(* IEC 61131-3 sources: com.logicals.lc3.webinar/usRTS_RPMControl_iSOC/src_FB_LIB_SAFE/Safe/PLCOpen (part 2) *)

(* ---- SF_GuardLocking_2.iecst ---- *)
USING logicals.web.standard.safe;

NAMESPACE logicals.web.standard.safe
NAMESPACE plcopen

TYPE
	SF_GuardLocking_2_State : UINT(
		/* Static Reset detected in state 8x01. */
		Reset_Error_0 := 16#C001,
		/* S_GuardLock and S_Guard are not TRUE although the door was not re-quested to be opened. */
		Guard_Error := 16#C010,
		/* Static Reset detected in state C410. */
		Reset_Error_1 := 16#C011,
		/* S_GuardLock and S_Guard become TRUE again after being lost (C010) */
		Guard_Return := 16#C410,
		/* Lost safety acknowledge signal. S_Guard and S_GuardLock are TRUE. */
		Safety_Lost_S_Guard_And_S_GuardLock_True := 16#C450,
		/* Lost safety acknowledge signal. At least one of the variables S_Guard or S_GuardLock is FALSE. */
		Safety_Lost_S_Guard_Or_S_GuardLock_False := 16#C050,
		/* Static Reset detected in state C420. */
		Reset_Error_2 := 16#C021,
		/* Safety acknowledge signal becomes TRUE again after being lost (Cx50). */
		Safety_Return := 16#C420,
		/* Static Reset detected in state 8433. */
		Reset_Error_3 := 16#C031,
		/* Waiting time to Unlock exceeded. */
		Unlock_Request_Error := 16#C440,
		/* Static Reset detected in state C440. */
		Reset_Error_4 := 16#C041,
		/* The function block is not active (initial state). */
		Idle := 16#0000,
		/* Guard is closed and locked. */
		Guard_Closed_And_Locked:= 16#8000,
		/* Function block was activated and initiated. S_Guard and S_GuardLock are TRUE. */
		Init_S_Guard_And_S_GuardLock_True := 16#8401,
		/* Function block was activated and initiated. At least one of the variables S_Guard or S_GuardLock is FALSE. */
		Init_S_Guard_Or_S_GuardLock_False := 16#8801,
		/* Door is closed and locked, now waiting for operator reset */
		Wait_For_Reset := 16#8430,
		/* Waiting for operator to request to open the door (unlock request). */
		Wait_For_Operator := 16#8812,
		/* Lock is released and guard is open. */
		Guard_Open_And_Unlocked := 16#8822,
		/* Lock is released but guard is closed. */
		Guard_Closed_But_Unlocked := 16#8832,
		/* S_UnlockGuard is TRUE, however the acknowledge signal S_GuardLocked is still TRUE (so waiting for acknowledge <FALSE>) */
		Wait_For_Unlocked := 16#8010
	);
END_TYPE

/* This FB controls an entrance to a hazardous area via an interlocking guard with guard locking ("four state interlock-ing"). */
FUNCTION_BLOCK SF_GuardLocking_2
	{ altName:="SF_GuardLocking_2"; bgColor:="Gold"; width:=400; }
	VAR_INPUT
		/* See 5.1.1 General Input Parameters */
		Activate : BOOL := FALSE;
		/* Variable.
		 * Monitors the guard interlocking. Can be connected to the GuardOut of the SF_Guard FB.
		 * FALSE: Guard open.
		 * TRUE: Guard closed and guarded area safe. */
		S_Guard : SAFEBOOL := SAFEBOOL_Constant#SAFEFALSE;
		/* Variable.
		 * Status of the hazardous area (EDM), e.g., based on speed moni-toring or safe time off delay.
		 * FALSE: Machine in "non-safe" state.
		 * TRUE: Machine in safe state. */
		S_SafetyActive : SAFEBOOL := SAFEBOOL_Constant#SAFEFALSE;
		/* Variable.
		 * Status of the mechanical guard locking.
		 * FALSE: Guard is not locked.
		 * TRUE: Guard is locked. */
		S_GuardLock : SAFEBOOL := SAFEBOOL_Constant#SAFEFALSE;
		/* Variable.
		 * Operator intervention - request to unlock the guard.
		 * FALSE: No request.
		 * TRUE: Request made. */
		UnlockRequest : BOOL := FALSE;
		/* See 5.1.1 General Input Parameters */
		S_StartReset : SAFEBOOL := SAFEBOOL_Constant#SAFEFALSE;
		/* See 5.1.1 General Input Parameters */
		S_AutoReset : SAFEBOOL := SAFEBOOL_Constant#SAFEFALSE;
		/* See 5.1.1 General Input Parameters.
		 * Also used to request the guard to be locked again.
		 * The quality of the signal must con-form to a manual reset device. */
		Reset : BOOL := FALSE;
	END_VAR

	VAR_OUTPUT
		/* See 5.1.2 General Output Parameters */
		Ready : BOOL := FALSE;
		/* Interface to hazardous area which must be stopped.
		 * FALSE: No safe state.
		 * TRUE: Safe state. */
		S_GuardLocked : SAFEBOOL := SAFEBOOL_Constant#SAFEFALSE;
		/* Signal to unlock the guard.
		 * FALSE: Close guard.
		 * TRUE: Unlock guard. */
		S_UnlockGuard : SAFEBOOL := SAFEBOOL_Constant#SAFEFALSE;
		/* Optional. See 5.1.2 General Output Parameters */
		SafetyDemand : BOOL := FALSE;
		/* Optional. See 5.1.2 General Output Parameters */
		ResetRequest : BOOL := FALSE;
		/* See 5.1.2 General Output Parameters */
		Error : BOOL := FALSE;
		/* See 5.1.2 General Output Parameters */
		DiagCode : WORD := 16#0000;
	END_VAR

	VAR
		R_Trig_Reset : R_TRIG;
		R_Trig_UnlockRequest : R_TRIG;
		Unlock_Waiting_Timer : TON;
	END_VAR

	R_Trig_Reset(Reset);
	R_Trig_UnlockRequest(UnlockRequest);

	IF(NOT Activate) THEN
		DiagCode := TO_WORD(SF_GuardLocking_2_State#Idle);
	ELSE
		CASE TO_UINT(DiagCode) OF
			SF_GuardLocking_2_State#Idle:
				/* IF(Activate) THEN - Active is always true here */
				IF(IS(S_Guard) AND IS(S_GuardLock)) THEN
					DiagCode := TO_WORD(SF_GuardLocking_2_State#Init_S_Guard_And_S_GuardLock_True);
				ELSE
					DiagCode := TO_WORD(SF_GuardLocking_2_State#Init_S_Guard_Or_S_GuardLock_False);
				END_IF;
			SF_GuardLocking_2_State#Init_S_Guard_And_S_GuardLock_True,
			SF_GuardLocking_2_State#Init_S_Guard_Or_S_GuardLock_False:
				IF(Reset AND NOT R_Trig_Reset.Q AND IS_NOT(S_StartReset)) THEN
					DiagCode := TO_WORD(SF_GuardLocking_2_State#Reset_Error_0);
				ELSIF(IS_NOT(S_Guard) AND UnlockRequest) THEN
					DiagCode := TO_WORD(SF_GuardLocking_2_State#Guard_Open_And_Unlocked);
				ELSIF(IS_NOT(S_Guard) AND NOT UnlockRequest) THEN
					DiagCode := TO_WORD(SF_GuardLocking_2_State#Guard_Error);
				ELSIF((R_Trig_Reset.Q OR IS(S_StartReset)) AND IS(S_Guard) AND IS(S_GuardLock)) THEN
					DiagCode := TO_WORD(SF_GuardLocking_2_State#Guard_Closed_And_Locked);
				END_IF;
			SF_GuardLocking_2_State#Reset_Error_0:
				IF(NOT Reset) THEN
					IF(IS(S_Guard) AND IS(S_GuardLock)) THEN
						DiagCode := TO_WORD(SF_GuardLocking_2_State#Init_S_Guard_And_S_GuardLock_True);
					ELSE
						DiagCode := TO_WORD(SF_GuardLocking_2_State#Init_S_Guard_Or_S_GuardLock_False);
					END_IF;
				END_IF;
			SF_GuardLocking_2_State#Guard_Open_And_Unlocked:
				IF(IS_NOT(S_SafetyActive)) THEN
					DiagCode := DetermineSafetyLost_GuardLocking_2(S_Guard, S_GuardLock);
				ELSIF(IS(S_Guard)) THEN
					DiagCode := TO_WORD(SF_GuardLocking_2_State#Guard_Closed_But_Unlocked);
				END_IF;
			SF_GuardLocking_2_State#Safety_Lost_S_Guard_And_S_GuardLock_True,
			SF_GuardLocking_2_State#Safety_Lost_S_Guard_Or_S_GuardLock_False:
				IF(IS(S_SafetyActive)) THEN
					DiagCode := TO_WORD(SF_GuardLocking_2_State#Safety_Return);
				ELSIF(R_Trig_Reset.Q AND IS(S_GuardLock) AND IS(S_Guard)) THEN
					DiagCode := TO_WORD(SF_GuardLocking_2_State#Guard_Closed_And_Locked);
				END_IF;
			SF_GuardLocking_2_State#Safety_Return:
				IF(Reset AND NOT R_Trig_Reset.Q) THEN
					DiagCode := TO_WORD(SF_GuardLocking_2_State#Reset_Error_2);
				ELSIF(IS_NOT(S_SafetyActive)) THEN
					DiagCode := DetermineSafetyLost_GuardLocking_2(S_Guard, S_GuardLock);
				ELSIF(R_Trig_Reset.Q AND (IS_NOT(S_GuardLock) OR IS_NOT(S_Guard))) THEN
					DiagCode := TO_WORD(SF_GuardLocking_2_State#Wait_For_Operator);
				ELSIF(R_Trig_Reset.Q AND IS(S_GuardLock) AND IS(S_Guard)) THEN
					DiagCode := TO_WORD(SF_GuardLocking_2_State#Guard_Closed_And_Locked);
				END_IF;
			SF_GuardLocking_2_State#Reset_Error_2:
				IF(NOT Reset) THEN
					DiagCode := TO_WORD(SF_GuardLocking_2_State#Safety_Return);
				END_IF;
			SF_GuardLocking_2_State#Guard_Closed_But_Unlocked:
				IF(IS_NOT(S_SafetyActive)) THEN
					DiagCode := DetermineSafetyLost_GuardLocking_2(S_Guard, S_GuardLock);
				ELSIF(IS_NOT(S_Guard)) THEN
					DiagCode := TO_WORD(SF_GuardLocking_2_State#Guard_Open_And_Unlocked);
				ELSIF(NOT UnlockRequest) THEN
					DiagCode := TO_WORD(SF_GuardLocking_2_State#Wait_For_Operator);
				END_IF;
			SF_GuardLocking_2_State#Wait_For_Operator:
				IF(IS_NOT(S_SafetyActive)) THEN
					DiagCode := DetermineSafetyLost_GuardLocking_2(S_Guard, S_GuardLock);
				ELSIF((IS(S_SafetyActive) AND UnlockRequest) OR IS_NOT(S_Guard)) THEN
					DiagCode := TO_WORD(SF_GuardLocking_2_State#Guard_Open_And_Unlocked);
				ELSIF(IS(S_Guard) AND IS(S_GuardLock) AND IS_NOT(S_AutoReset)) THEN
					DiagCode := TO_WORD(SF_GuardLocking_2_State#Wait_For_Reset);
				ELSIF(IS(S_Guard) AND IS(S_GuardLock) AND IS(S_AutoReset)) THEN
					DiagCode := TO_WORD(SF_GuardLocking_2_State#Guard_Closed_And_Locked);
				END_IF;
			SF_GuardLocking_2_State#Wait_For_Reset:
				IF(Reset AND NOT R_Trig_Reset.Q) THEN
					DiagCode := TO_WORD(SF_GuardLocking_2_State#Reset_Error_3);
				ELSIF(IS_NOT(S_Guard) OR IS_NOT(S_GuardLock)) THEN
					DiagCode := TO_WORD(SF_GuardLocking_2_State#Guard_Error);
				ELSIF(R_Trig_Reset.Q) THEN
					DiagCode := TO_WORD(SF_GuardLocking_2_State#Guard_Closed_And_Locked);
				ELSIF(R_Trig_UnlockRequest.Q) THEN
					DiagCode := TO_WORD(SF_GuardLocking_2_State#Wait_For_Unlocked);
				END_IF;
			SF_GuardLocking_2_State#Reset_Error_3:
				IF(NOT Reset) THEN
					DiagCode := TO_WORD(SF_GuardLocking_2_State#Wait_For_Reset);
				END_IF;
			SF_GuardLocking_2_State#Guard_Error:
				IF(IS(S_GuardLock) AND IS(S_Guard)) THEN
					DiagCode := TO_WORD(SF_GuardLocking_2_State#Guard_Return);
				END_IF;
			SF_GuardLocking_2_State#Guard_Return:
				IF(IS_NOT(S_GuardLock) OR IS_NOT(S_Guard)) THEN
					DiagCode := TO_WORD(SF_GuardLocking_2_State#Guard_Error);
				ELSIF(Reset AND NOT R_Trig_Reset.Q) THEN
					DiagCode := TO_WORD(SF_GuardLocking_2_State#Reset_Error_1);
				ELSIF(R_Trig_Reset.Q) THEN
					DiagCode := TO_WORD(SF_GuardLocking_2_State#Guard_Closed_And_Locked);
				END_IF;
			SF_GuardLocking_2_State#Reset_Error_1:
				IF(NOT Reset) THEN
					DiagCode := TO_WORD(SF_GuardLocking_2_State#Guard_Return);
				END_IF;
			SF_GuardLocking_2_State#Wait_For_Unlocked:
				Unlock_Waiting_Timer();
				IF(IS_NOT(S_SafetyActive)) THEN
					DiagCode := DetermineSafetyLost_GuardLocking_2(S_Guard, S_GuardLock);
				ELSIF(IS_NOT(S_GuardLock)) THEN
					DiagCode := TO_WORD(SF_GuardLocking_2_State#Guard_Closed_But_Unlocked);
				ELSIF(Unlock_Waiting_Timer.Q) THEN
					DiagCode := TO_WORD(SF_GuardLocking_2_State#Unlock_Request_Error);
				END_IF;
			SF_GuardLocking_2_State#Unlock_Request_Error:
				IF(Reset AND NOT R_Trig_Reset.Q) THEN
					DiagCode := TO_WORD(SF_GuardLocking_2_State#Reset_Error_4);
				ELSIF(IS_NOT(S_Guard) OR IS_NOT(S_GuardLock)) THEN
					DiagCode := TO_WORD(SF_GuardLocking_2_State#Guard_Error);
				ELSIF(R_Trig_Reset.Q AND IS(S_GuardLock) AND IS(S_Guard)) THEN
					DiagCode := TO_WORD(SF_GuardLocking_2_State#Guard_Closed_And_Locked);
				END_IF;
			SF_GuardLocking_2_State#Reset_Error_4:
				IF(NOT Reset) THEN
					DiagCode := TO_WORD(SF_GuardLocking_2_State#Unlock_Request_Error);
				END_IF;
			SF_GuardLocking_2_State#Guard_Closed_And_Locked:
				IF(IS_NOT(S_GuardLock) OR IS_NOT(S_Guard)) THEN
					DiagCode := TO_WORD(SF_GuardLocking_2_State#Guard_Error);
				ELSIF(R_Trig_UnlockRequest.Q AND IS(S_SafetyActive)) THEN
					DiagCode := TO_WORD(SF_GuardLocking_2_State#Wait_For_Unlocked);
				END_IF;
		END_CASE;
	END_IF;

	CASE TO_UINT(DiagCode) OF
		SF_GuardLocking_2_State#Reset_Error_0,
		SF_GuardLocking_2_State#Guard_Error,
		SF_GuardLocking_2_State#Reset_Error_1,
		SF_GuardLocking_2_State#Reset_Error_3:
			Unlock_Waiting_Timer(IN := FALSE);
			Ready := TRUE;
			S_GuardLocked := SAFEBOOL_Constant#SAFEFALSE;
			S_UnlockGuard := SAFEBOOL_Constant#SAFEFALSE;
			SafetyDemand := FALSE;
			ResetRequest := FALSE;
			Error := TRUE;
		SF_GuardLocking_2_State#Guard_Return:
			Unlock_Waiting_Timer(IN := FALSE);
			Ready := TRUE;
			S_GuardLocked := SAFEBOOL_Constant#SAFEFALSE;
			S_UnlockGuard := SAFEBOOL_Constant#SAFEFALSE;
			SafetyDemand := FALSE;
			ResetRequest := TRUE;
			Error := TRUE;
		SF_GuardLocking_2_State#Safety_Lost_S_Guard_And_S_GuardLock_True,
		SF_GuardLocking_2_State#Safety_Return,
		SF_GuardLocking_2_State#Unlock_Request_Error:
			Unlock_Waiting_Timer(IN := FALSE);
			Ready := TRUE;
			S_GuardLocked := SAFEBOOL_Constant#SAFEFALSE;
			S_UnlockGuard := SAFEBOOL_Constant#SAFETRUE;
			SafetyDemand := FALSE;
			ResetRequest := TRUE;
			Error := TRUE;
		SF_GuardLocking_2_State#Safety_Lost_S_Guard_Or_S_GuardLock_False,
		SF_GuardLocking_2_State#Reset_Error_2,
		SF_GuardLocking_2_State#Reset_Error_4:
			Unlock_Waiting_Timer(IN := FALSE);
			Ready := TRUE;
			S_GuardLocked := SAFEBOOL_Constant#SAFEFALSE;
			S_UnlockGuard := SAFEBOOL_Constant#SAFETRUE;
			SafetyDemand := FALSE;
			ResetRequest := FALSE;
			Error := TRUE;
		SF_GuardLocking_2_State#Idle:
			Unlock_Waiting_Timer(IN := FALSE);
			Ready := FALSE;
			S_GuardLocked := SAFEBOOL_Constant#SAFEFALSE;
			S_UnlockGuard := SAFEBOOL_Constant#SAFEFALSE;
			SafetyDemand := FALSE;
			ResetRequest := FALSE;
			Error := FALSE;
		SF_GuardLocking_2_State#Guard_Closed_And_Locked:
			Unlock_Waiting_Timer(IN := FALSE);
			Ready := TRUE;
			S_GuardLocked := SAFEBOOL_Constant#SAFETRUE;
			S_UnlockGuard := SAFEBOOL_Constant#SAFEFALSE;
			SafetyDemand := FALSE;
			ResetRequest := FALSE;
			Error := FALSE;
		SF_GuardLocking_2_State#Init_S_Guard_And_S_GuardLock_True,
		SF_GuardLocking_2_State#Wait_For_Reset:
			Unlock_Waiting_Timer(IN := FALSE);
			Ready := TRUE;
			S_GuardLocked := SAFEBOOL_Constant#SAFEFALSE;
			S_UnlockGuard := SAFEBOOL_Constant#SAFEFALSE;
			SafetyDemand := FALSE;
			ResetRequest := TRUE;
			Error := FALSE;
		SF_GuardLocking_2_State#Init_S_Guard_Or_S_GuardLock_False,
		SF_GuardLocking_2_State#Wait_For_Operator:
			Unlock_Waiting_Timer(IN := FALSE);
			Ready := TRUE;
			S_GuardLocked := SAFEBOOL_Constant#SAFEFALSE;
			S_UnlockGuard := SAFEBOOL_Constant#SAFEFALSE;
			SafetyDemand := TRUE;
			ResetRequest := FALSE;
			Error := FALSE;
		SF_GuardLocking_2_State#Guard_Open_And_Unlocked,
		SF_GuardLocking_2_State#Guard_Closed_But_Unlocked:
			Unlock_Waiting_Timer(IN := FALSE);
			Ready := TRUE;
			S_GuardLocked := SAFEBOOL_Constant#SAFEFALSE;
			S_UnlockGuard := SAFEBOOL_Constant#SAFETRUE;
			SafetyDemand := TRUE;
			ResetRequest := FALSE;
			Error := FALSE;
		SF_GuardLocking_2_State#Wait_For_Unlocked:
			Unlock_Waiting_Timer(IN := TRUE, PT := T#2s);
			Ready := TRUE;
			S_GuardLocked := SAFEBOOL_Constant#SAFEFALSE;
			S_UnlockGuard := SAFEBOOL_Constant#SAFETRUE;
			SafetyDemand := FALSE;
			ResetRequest := FALSE;
			Error := FALSE;
		ELSE
			ENO := FALSE;
	END_CASE;

	ENO := ENO AND CheckSAFEBOOL(S_Guard) AND CheckSAFEBOOL(S_SafetyActive) AND CheckSAFEBOOL(S_GuardLock) AND CheckSAFEBOOL(S_StartReset) AND CheckSAFEBOOL(S_AutoReset);

END_FUNCTION_BLOCK

FUNCTION DetermineSafetyLost_GuardLocking_2 : WORD
	VAR_INPUT
		S_Guard : SAFEBOOL;
		S_GuardLock : SAFEBOOL;
	END_VAR

	IF(IS(S_Guard) AND IS(S_GuardLock)) THEN
		DetermineSafetyLost_GuardLocking_2 := TO_WORD(SF_GuardLocking_2_State#Safety_Lost_S_Guard_And_S_GuardLock_True);
	ELSE
		DetermineSafetyLost_GuardLocking_2 := TO_WORD(SF_GuardLocking_2_State#Safety_Lost_S_Guard_Or_S_GuardLock_False);
	END_IF;
END_FUNCTION

END_NAMESPACE
END_NAMESPACE

(* ---- SF_GuardLockingSerial.iecst ---- *)
USING logicals.web.standard.safe;

NAMESPACE logicals.web.standard.safe
NAMESPACE plcopen

TYPE
	SF_GuardLockingSerial_State : UINT(
	/* Static Reset detected in state 8001. */
	Reset_Error_0 := 16#C001,
	/* S_Guard is not TRUE although the door was not requested to be opened. */
	Guard_Error := 16#C010,
	/* Static Reset detected in state C410. */
	Reset_Error_1 := 16#C011,
	/* S_Guard becomes TRUE again after being lost (C010). */
	Guard_Return := 16#C410,
	/* Lost safety acknowledge signal. S_Guard is TRUE. */
	Safety_Lost_S_Guard_True := 16#C450,
	/* Lost safety acknowledge signal. S_Guard is FALSE. */
	Safety_Lost_S_Guard_False := 16#C050,
	/* Static Reset detected in state C420. */
	Reset_Error_2 := 16#C021,
	/* Safety acknowledge signal becomes TRUE again after being lost (Cx50). */
	Safety_Return := 16#C420,
	/* Static Reset detected in state 8430. */
	Reset_Error_3 := 16#C031,
	/* Waiting time to Unlock exceeded. S_Guard is TRUE. */
	Unlock_Request_Error_S_Guard_True := 16#C440,
	/* Waiting time to Unlock exceeded. S_Guard is FALSE. */
	Unlock_Request_Error_S_Guard_False := 16#C040,
	/* Static Reset detected in state Cx40. */
	Reset_Error_4 := 16#C041,
	/* The function block is not active (initial state). */
	Idle := 16#0000,
	/* Guard is closed and locked. */
	Guard_Closed_And_Locked := 16#8000,
	/* Function block was activated and initiated. S_Guard is TRUE. */
	Init_S_Guard_True := 16#8401,
	/* Function block was activated and initiated. S_Guard is FALSE. */
	Init_S_Guard_False := 16#8801,
	/* Door is closed and locked, now waiting for operator reset */
	Wait_For_Reset := 16#8430,
	/* Waiting for operator to request to open the door (unlock request). */
	Wait_For_Operator := 16#8812,
	/* Guard is unlocked. Door can be closed or open. */
	Guard_Open_And_Or_Unlocked := 16#8822,
	/* S_UnlockGuard is TRUE, however the acknowledge signal S_GuardLocked is still TRUE (so waiting for acknowledge <FALSE>) */
	Wait_For_Unlocked := 16#8410
	);
END_TYPE

/*
 * This FB controls an entrance to a hazardous area via an interlocking guard with guard locking (four state interlock-ing).
 * The used switch does not distinguish between if the safety door is unlocked but not opened or unlocked and opened.
 * Therefore we only have the S_Guard input compared to SF_GuardLocking_2.
 */
FUNCTION_BLOCK SF_GuardLockingSerial
	{ altName:="SF_GuardLockingSerial"; bgColor:="Gold"; width:=420; }
	VAR_INPUT
		/* See 5.1.1 General Input Parameters */
		Activate : BOOl := FALSE;
		/* Variable.
		 * Monitors the guard interlocking. This can be connect to S_GuardOut from the SF_Guard FB
		 * FALSE: Guard open.
		 * TRUE: Guard closed and guarded area safe. */
		S_Guard : SAFEBOOL := SAFEBOOL_Constant#SAFEFALSE;
		/* Variable.
		 * Status of the hazardous area (EDM), e.g., based on speed moni-toring or safe time off delay.
		 * FALSE: Machine in "non-safe" state.
		 * TRUE: Machine in safe state. */
		S_SafetyActive : SAFEBOOL := SAFEBOOL_Constant#SAFEFALSE;
		/* Variable.
		 * Operator intervention  request to unlock the guard.
		 * FALSE: No request.
		 * TRUE: Request made. */
		UnlockRequest : BOOL := FALSE;
		/* See 5.1.1 General Input Parameters */
		S_StartReset : SAFEBOOL := SAFEBOOL_Constant#SAFEFALSE;
		/* See 5.1.1 General Input Parameters */
		S_AutoReset : SAFEBOOL := SAFEBOOL_Constant#SAFEFALSE;
		/* See 5.1.1 General Input Parameters.
		 * Also used to request the guard to be locked again. The quality of the signal must conform to a manual reset device. */
		Reset : BOOL := FALSE;
	END_VAR

	VAR_OUTPUT
		/* See 5.1.2 General Output Parameters */
		Ready : BOOL := FALSE;
		/* Interface to hazardous area which must be stopped.
		 * FALSE: No safe state.
		 * TRUE: Safe state. */
		S_GuardLocked : SAFEBOOL := SAFEBOOL_Constant#SAFEFALSE;
		/* Signal to unlock the guard.
		 * FALSE: Close guard.
		 * TRUE: Unlock guard. */
		S_UnlockGuard : SAFEBOOL := SAFEBOOL_Constant#SAFEFALSE;
		/* See 5.1.2 General Output Parameters */
		SafetyDemand : BOOL := FALSE;
		/* See 5.1.2 General Output Parameters */
		ResetRequest : BOOL := FALSE;
		/* See 5.1.2 General Output Parameters */
		Error : BOOL := FALSE;
		/* See 5.1.2 General Output Parameters */
		DiagCode : WORD := 16#0000;
	END_VAR

	VAR
		R_Trig_Reset : R_TRIG;
		R_Trig_UnlockRequest : R_TRIG;
		Unlock_Waiting_Timer : TON;
	END_VAR

	R_Trig_Reset(Reset);
	R_Trig_UnlockRequest(UnlockRequest);

	IF(NOT Activate) THEN
		DiagCode := TO_WORD(SF_GuardLockingSerial_State#Idle);
	ELSE
		CASE TO_UINT(DiagCode) OF
			SF_GuardLockingSerial_State#Idle:
				/* IF(Activate) THEN - Active is always true here */
				IF(IS(S_Guard)) THEN
					DiagCode := TO_WORD(SF_GuardLockingSerial_State#Init_S_Guard_True);
				ELSE
					DiagCode := TO_WORD(SF_GuardLockingSerial_State#Init_S_Guard_False);
				END_IF;
			SF_GuardLockingSerial_State#Init_S_Guard_True,
			SF_GuardLockingSerial_State#Init_S_Guard_False:
				IF(Reset AND NOT R_Trig_Reset.Q AND IS_NOT(S_StartReset)) THEN
					DiagCode := TO_WORD(SF_GuardLockingSerial_State#Reset_Error_0);
				ELSIF(IS_NOT(S_Guard) AND UnlockRequest) THEN
					DiagCode := TO_WORD(SF_GuardLockingSerial_State#Guard_Open_And_Or_Unlocked);
				ELSIF(IS_NOT(S_Guard) AND NOT UnlockRequest) THEN
					DiagCode := TO_WORD(SF_GuardLockingSerial_State#Guard_Error);
				ELSIF((R_Trig_Reset.Q OR IS(S_StartReset)) AND IS(S_Guard)) THEN
					DiagCode := TO_WORD(SF_GuardLockingSerial_State#Guard_Closed_And_Locked);
				END_IF;
			SF_GuardLockingSerial_State#Guard_Open_And_Or_Unlocked:
				IF(IS_NOT(S_SafetyActive)) THEN
					DiagCode := DetermineSafetyLost_GuardLockingSerial(S_Guard);
				ELSIF(NOT UnlockRequest) THEN
					DiagCode := TO_WORD(SF_GuardLockingSerial_State#Wait_For_Operator);
				END_IF;
			SF_GuardLockingSerial_State#Safety_Lost_S_Guard_True,
			SF_GuardLockingSerial_State#Safety_Lost_S_Guard_False:
				IF(IS(S_SafetyActive)) THEN
					DiagCode := TO_WORD(SF_GuardLockingSerial_State#Safety_Return);
				ELSIF(R_Trig_Reset.Q AND IS(S_Guard)) THEN
					DiagCode := TO_WORD(SF_GuardLockingSerial_State#Guard_Closed_And_Locked);
				END_IF;
			SF_GuardLockingSerial_State#Safety_Return:
				IF(Reset AND NOT R_Trig_Reset.Q) THEN
					DiagCode := TO_WORD(SF_GuardLockingSerial_State#Reset_Error_2);
				ELSIF(IS_NOT(S_SafetyActive)) THEN
					DiagCode := DetermineSafetyLost_GuardLockingSerial(S_Guard);
				ELSIF(R_Trig_Reset.Q AND IS_NOT(S_Guard)) THEN
					DiagCode := TO_WORD(SF_GuardLockingSerial_State#Wait_For_Operator);
				ELSIF(R_Trig_Reset.Q AND IS(S_Guard)) THEN
					DiagCode := TO_WORD(SF_GuardLockingSerial_State#Guard_Closed_And_Locked);
				END_IF;
			SF_GuardLockingSerial_State#Wait_For_Operator:
				IF(IS_NOT(S_SafetyActive)) THEN
					DiagCode := DetermineSafetyLost_GuardLockingSerial(S_Guard);
				//NOTE: This transition was adapted, because when using the original transition, transition 3 would be unreachable!
				ELSIF(IS(S_Guard) AND IS_NOT(S_AutoReset)) THEN
					DiagCode := TO_WORD(SF_GuardLockingSerial_State#Wait_For_Reset);
				ELSIF(IS(S_Guard) AND IS(S_AutoReset)) THEN
					DiagCode := TO_WORD(SF_GuardLockingSerial_State#Guard_Closed_And_Locked);
				END_IF;
			SF_GuardLockingSerial_State#Wait_For_Reset:
				IF(Reset AND NOT R_Trig_Reset.Q AND IS_NOT(S_AutoReset)) THEN
					DiagCode := TO_WORD(SF_GuardLockingSerial_State#Reset_Error_3);
				ELSIF(IS_NOT(S_Guard)) THEN
					DiagCode := TO_WORD(SF_GuardLockingSerial_State#Guard_Error);
				ELSIF(R_Trig_Reset.Q) THEN
					DiagCode := TO_WORD(SF_GuardLockingSerial_State#Guard_Closed_And_Locked);
				ELSIF(R_Trig_UnlockRequest.Q) THEN
					DiagCode := TO_WORD(SF_GuardLockingSerial_State#Wait_For_Unlocked);
				END_IF;
			SF_GuardLockingSerial_State#Wait_For_Unlocked:
				Unlock_Waiting_Timer();
				IF(IS_NOT(S_Guard)) THEN
					DiagCode := TO_WORD(SF_GuardLockingSerial_State#Guard_Open_And_Or_Unlocked);
				ELSIF(R_Trig_Reset.Q AND IS(S_Guard)) THEN
					DiagCode := TO_WORD(SF_GuardLockingSerial_State#Guard_Closed_And_Locked);
				ELSIF(Unlock_Waiting_Timer.Q) THEN
					//S_Guard can only be TRUE here -> no need to check it
					DiagCode := TO_WORD(SF_GuardLockingSerial_State#Unlock_Request_Error_S_Guard_True);
				END_IF;
			SF_GuardLockingSerial_State#Unlock_Request_Error_S_Guard_True,
			SF_GuardLockingSerial_State#Unlock_Request_Error_S_Guard_False:
				IF(Reset AND NOT R_Trig_Reset.Q AND IS_NOT(S_AutoReset)) THEN
					DiagCode := TO_WORD(SF_GuardLockingSerial_State#Reset_Error_4);
				ELSIF(R_Trig_Reset.Q AND IS(S_Guard)) THEN
					DiagCode := TO_WORD(SF_GuardLockingSerial_State#Guard_Closed_And_Locked);
				END_IF;
			SF_GuardLockingSerial_State#Guard_Closed_And_Locked:
				IF(IS_NOT(S_Guard)) THEN
					DiagCode := TO_WORD(SF_GuardLockingSerial_State#Guard_Error);
				ELSIF(R_Trig_UnlockRequest.Q AND IS(S_SafetyActive)) THEN
					DiagCode := TO_WORD(SF_GuardLockingSerial_State#Wait_For_Unlocked);
				END_IF;
			SF_GuardLockingSerial_State#Guard_Error:
				IF(IS(S_Guard)) THEN
					DiagCode := TO_WORD(SF_GuardLockingSerial_State#Guard_Return);
				END_IF;
			SF_GuardLockingSerial_State#Guard_Return:
				IF(IS_NOT(S_Guard)) THEN
					DiagCode := TO_WORD(SF_GuardLockingSerial_State#Guard_Error);
				ELSIF(Reset AND NOT R_Trig_Reset.Q) THEN
					DiagCode := TO_WORD(SF_GuardLockingSerial_State#Reset_Error_1);
				ELSIF(R_Trig_Reset.Q AND IS(S_Guard)) THEN
					DiagCode := TO_WORD(SF_GuardLockingSerial_State#Guard_Closed_And_Locked);
				END_IF;
			SF_GuardLockingSerial_State#Reset_Error_0:
				IF(NOT Reset) THEN
					IF(IS(S_Guard)) THEN
						DiagCode := TO_WORD(SF_GuardLockingSerial_State#Init_S_Guard_True);
					ELSE
						DiagCode := TO_WORD(SF_GuardLockingSerial_State#Init_S_Guard_False);
					END_IF;
				END_IF;
			SF_GuardLockingSerial_State#Reset_Error_1:
				IF(NOT Reset) THEN
					DiagCode := TO_WORD(SF_GuardLockingSerial_State#Guard_Return);
				END_IF;
			SF_GuardLockingSerial_State#Reset_Error_2:
				IF(NOT Reset) THEN
					DiagCode := TO_WORD(SF_GuardLockingSerial_State#Safety_Return);
				END_IF;
			SF_GuardLockingSerial_State#Reset_Error_3:
				IF(NOT Reset) THEN
					DiagCode := TO_WORD(SF_GuardLockingSerial_State#Wait_For_Reset);
				END_IF;
			SF_GuardLockingSerial_State#Reset_Error_4:
				IF(NOT Reset) THEN
					IF(IS(S_Guard)) THEN
						DiagCode := TO_WORD(SF_GuardLockingSerial_State#Unlock_Request_Error_S_Guard_True);
					ELSE
						DiagCode := TO_WORD(SF_GuardLockingSerial_State#Unlock_Request_Error_S_Guard_False);
					END_IF;
				END_IF;
		END_CASE;
	END_IF;

	CASE TO_UINT(DiagCode) OF
		SF_GuardLockingSerial_State#Idle:
			Unlock_Waiting_Timer(IN := FALSE);
			Ready := FALSE;
			S_GuardLocked := SAFEBOOL_Constant#SAFEFALSE;
			S_UnlockGuard := SAFEBOOL_Constant#SAFEFALSE;
			SafetyDemand := FALSE;
			ResetRequest := FALSE;
			Error := FALSE;
		SF_GuardLockingSerial_State#Guard_Closed_And_Locked:
			Unlock_Waiting_Timer(IN := FALSE);
			Ready := TRUE;
			S_GuardLocked := SAFEBOOL_Constant#SAFETRUE;
			S_UnlockGuard := SAFEBOOL_Constant#SAFEFALSE;
			SafetyDemand := FALSE;
			ResetRequest := FALSE;
			Error := FALSE;
		SF_GuardLockingSerial_State#Init_S_Guard_True,
		SF_GuardLockingSerial_State#Wait_For_Reset:
			Unlock_Waiting_Timer(IN := FALSE);
			Ready := TRUE;
			S_GuardLocked := SAFEBOOL_Constant#SAFEFALSE;
			S_UnlockGuard := SAFEBOOL_Constant#SAFEFALSE;
			SafetyDemand := FALSE;
			ResetRequest := TRUE;
			Error := FALSE;
		SF_GuardLockingSerial_State#Init_S_Guard_False,
		SF_GuardLockingSerial_State#Wait_For_Operator:
			Unlock_Waiting_Timer(IN := FALSE);
			Ready := TRUE;
			S_GuardLocked := SAFEBOOL_Constant#SAFEFALSE;
			S_UnlockGuard := SAFEBOOL_Constant#SAFEFALSE;
			SafetyDemand := TRUE;
			ResetRequest := FALSE;
			Error := FALSE;
		SF_GuardLockingSerial_State#Guard_Open_And_Or_Unlocked:
			Unlock_Waiting_Timer(IN := FALSE);
			Ready := TRUE;
			S_GuardLocked := SAFEBOOL_Constant#SAFEFALSE;
			S_UnlockGuard := SAFEBOOL_Constant#SAFETRUE;
			SafetyDemand := TRUE;
			ResetRequest := FALSE;
			Error := FALSE;
		SF_GuardLockingSerial_State#Wait_For_Unlocked:
			Unlock_Waiting_Timer(IN := TRUE, PT := T#2s);
			Ready := TRUE;
			S_GuardLocked := SAFEBOOL_Constant#SAFEFALSE;
			S_UnlockGuard := SAFEBOOL_Constant#SAFETRUE;
			SafetyDemand := FALSE;
			ResetRequest := TRUE;
			Error := FALSE;
		SF_GuardLockingSerial_State#Reset_Error_0,
		SF_GuardLockingSerial_State#Guard_Error,
		SF_GuardLockingSerial_State#Reset_Error_1,
		SF_GuardLockingSerial_State#Reset_Error_3:
			Unlock_Waiting_Timer(IN := FALSE);
			Ready := TRUE;
			S_GuardLocked := SAFEBOOL_Constant#SAFEFALSE;
			S_UnlockGuard := SAFEBOOL_Constant#SAFEFALSE;
			SafetyDemand := FALSE;
			ResetRequest := FALSE;
			Error := TRUE;
		SF_GuardLockingSerial_State#Guard_Return:
			Unlock_Waiting_Timer(IN := FALSE);
			Ready := TRUE;
			S_GuardLocked := SAFEBOOL_Constant#SAFEFALSE;
			S_UnlockGuard := SAFEBOOL_Constant#SAFEFALSE;
			SafetyDemand := FALSE;
			ResetRequest := TRUE;
			Error := TRUE;
		SF_GuardLockingSerial_State#Safety_Lost_S_Guard_True,
		SF_GuardLockingSerial_State#Safety_Return,
		SF_GuardLockingSerial_State#Unlock_Request_Error_S_Guard_True:
			 Unlock_Waiting_Timer(IN := FALSE);
			Ready := TRUE;
			S_GuardLocked := SAFEBOOL_Constant#SAFEFALSE;
			S_UnlockGuard := SAFEBOOL_Constant#SAFETRUE;
			SafetyDemand := FALSE;
			ResetRequest := TRUE;
			Error := TRUE;
		SF_GuardLockingSerial_State#Safety_Lost_S_Guard_False,
		SF_GuardLockingSerial_State#Reset_Error_2,
		SF_GuardLockingSerial_State#Unlock_Request_Error_S_Guard_False,
		SF_GuardLockingSerial_State#Reset_Error_4:
			Unlock_Waiting_Timer(IN := FALSE);
			Ready := TRUE;
			S_GuardLocked := SAFEBOOL_Constant#SAFEFALSE;
			S_UnlockGuard := SAFEBOOL_Constant#SAFETRUE;
			SafetyDemand := FALSE;
			ResetRequest := FALSE;
			Error := TRUE;
		ELSE
			ENO := FALSE;
	END_CASE;

	ENO := ENO AND CheckSAFEBOOL(S_Guard) AND CheckSAFEBOOL(S_SafetyActive) AND CheckSAFEBOOL(S_StartReset) AND CheckSAFEBOOL(S_AutoReset);
END_FUNCTION_BLOCK

FUNCTION DetermineSafetyLost_GuardLockingSerial : WORD
	VAR_INPUT
		S_Guard : SAFEBOOL;
	END_VAR

	IF(IS(S_Guard)) THEN
		DetermineSafetyLost_GuardLockingSerial := TO_WORD(SF_GuardLockingSerial_State#Safety_Lost_S_Guard_True);
	ELSE
		DetermineSafetyLost_GuardLockingSerial := TO_WORD(SF_GuardLockingSerial_State#Safety_Lost_S_Guard_False);
	END_IF;
END_FUNCTION

END_NAMESPACE
END_NAMESPACE

(* ---- SF_ModeSelector.iecst ---- *)
USING logicals.web.standard.safe;

NAMESPACE logicals.web.standard.safe
NAMESPACE plcopen

TYPE
	SF_ModeSelector_State : UINT(
	/* The FB detected that two or more S_ModeX are TRUE, e.g., short-circuit of cables. Only one S_ModeX OR no S_ModeX = TRUE */
	Error_Short_Circuit := 16#C010,
	Error_Short_Circuit_Fixed := 16#C410,

	/* The FB detected that all S_ModeX are FALSE: The period following a falling S_ModeX trigger exceeds ModeMonitorTime, e.g., open-circuit of cables. Only one S_ModeX = TRUE */
	Error_Open_Circuit := 16#C020,
	Error_Open_Circuit_Fixed := 16#C420,

	/* Static Reset signal detected in state C410. */
	Reset_Error_1 := 16#C011,
	/* Static Reset signal detected in state C420. */
	Reset_Error_2 := 16#C021,
	/* The function block is not active (initial state). */
	Idle := 16#0000,
	/* State after activation or when S_ModeX has changed (unless locked) or after Reset of an error state. */
	Mode_Changed := 16#8802,
	/* Valid mode selection, but not yet locked. */
	Mode_Selected := 16#8000,
	/* Valid mode selection is locked. */
	Mode_Locked := 16#8010
	);

	ModeState : INT(Only_One_S_ModeX := 0, No_S_ModeX := 1, More_Than_One_S_ModeX := 2);

END_TYPE

/* This function block selects the system operation mode, such as manual, automatic, semi-automatic, etc. */
FUNCTION_BLOCK SF_ModeSelector
	{ altName:="SF_ModeSelector"; bgColor:="Gold"; width:=340; }
	VAR_INPUT
		/* See Table 5.1.1 General Input Parameters */
		Activate : BOOL := FALSE;
		/* Variable or constant.
		* Input 0 from mode selector switch
		* FALSE: Mode 0 is not requested by operator.
		* TRUE: Mode 0 is requested by operator. */
		S_Mode0 : SAFEBOOL := SAFEBOOL_Constant#SAFEFALSE;
		/* Variable or constant.
		 * Input 1 from mode selector switch
		 * FALSE: Mode 1 is not requested by operator.
		 * TRUE: Mode 1 is requested by operator. */
		S_Mode1 : SAFEBOOL := SAFEBOOL_Constant#SAFEFALSE;
		/* Variable or constant.
		 * Input 2 from mode selector switch
		 * FALSE: Mode 2 is not requested by operator.
		 * TRUE: Mode 2 is requested by operator. */
		S_Mode2 : SAFEBOOL := SAFEBOOL_Constant#SAFEFALSE;
		/* Variable or constant.
		 * Input 3 from mode selector switch
		 * FALSE: Mode 3 is not requested by operator.
		 * TRUE: Mode 3 is requested by operator. */
		S_Mode3 : SAFEBOOL := SAFEBOOL_Constant#SAFEFALSE;
		/* Variable or constant.
		 * Input 4 from mode selector switch
		 * FALSE: Mode 4 is not requested by operator.
		 * TRUE: Mode 4 is requested by operator. */
		S_Mode4 : SAFEBOOL := SAFEBOOL_Constant#SAFEFALSE;
		/* Variable or constant.
		 * Input 5 from mode selector switch
		 * FALSE: Mode 5 is not requested by operator.
		 * TRUE: Mode 5 is requested by operator. */
		S_Mode5 : SAFEBOOL := SAFEBOOL_Constant#SAFEFALSE;
		/* Variable or constant.
		 * Input 6 from mode selector switch
		 * FALSE: Mode 6 is not requested by operator.
		 * TRUE: Mode 6 is requested by operator. */
		S_Mode6 : SAFEBOOL := SAFEBOOL_Constant#SAFEFALSE;
		/* Variable or constant.
		 * Input 7 from mode selector switch
		 * FALSE: Mode 7 is not requested by operator.
		 * TRUE: Mode 7 is requested by operator. */
		S_Mode7 : SAFEBOOL := SAFEBOOL_Constant#SAFEFALSE;
		/* Variable or constant.
		 * Locks the selected mode
		 * FALSE: The actual S_ModeXSel output is locked therefore a change of any S_ModeX input
		 * does not lead to a change in the S_ModeXSel output even in the event of a rising edge of Set-Mode.
		 * TRUE: The selected S_ModeXSel is not locked; a mode selec-tion change is possible. */
		S_Unlock : SAFEBOOL := SAFEBOOL_Constant#SAFEFALSE;
		/* Variable (or constant FALSE, if AutoSetMode = TRUE)
		 * Sets the selected mode
		 * Operator acknowledges the setting of a mode.
		 * Any change to new S_ModeX = TRUE leads to S_AnyModeSel/S_ModeXSel = FALSE, only a rising SetMode trigger then leads to new S_ModeXSel = TRUE. */
		S_SetMode : SAFEBOOL := SAFEBOOL_Constant#SAFEFALSE;
		/* Constant.
		 * Parameterizes the acknowledgement mode
		 * FALSE: A change in mode must be acknowledged by the operator via SetMode.
		 * TRUE: A valid change of the S_ModeX input to another S_ModeX automatically leads to a change in S_ModeXSel
		 * without operator acknowledgment via SetMode (as long as this is not locked by S_Unlock). */
		AutoSetMode : BOOL := FALSE;
		/* Constant.
		 * Maximum permissible time for changing the selection input. */
		ModeMonitorTime : TIME := T#0s;
		/* See Section 5.1.1 General Input Parameters */
		Reset : BOOL := FALSE;
	END_VAR

	VAR_OUTPUT
		/* See Section 5.1.2 General Output Parameters */
		Ready : BOOL := FALSE;
		/* Indicates that mode 0 is selected and acknowledged.
		 * FALSE: Mode 0 is not selected or not active.
		 * TRUE: Mode 0 is selected and active. */
		S_Mode0Sel : SAFEBOOL := FALSE;
		/* Indicates that mode 1 is selected and acknowledged.
		 * FALSE: Mode 1 is not selected or not active.
		 * TRUE: Mode 1 is selected and active. */
		S_Mode1Sel : SAFEBOOL := FALSE;
		/* Indicates that mode 2 is selected and acknowledged.
		 * FALSE: Mode 2 is not selected or not active.
		 * TRUE: Mode 2 is selected and active. */
		S_Mode2Sel : SAFEBOOL := FALSE;
		/* Indicates that mode 3 is selected and acknowledged.
		 * FALSE: Mode 3 is not selected or not active.
		 * TRUE: Mode 3 is selected and active. */
		S_Mode3Sel : SAFEBOOL := FALSE;
		/* Indicates that mode 4 is selected and acknowledged.
		 * FALSE: Mode 4 is not selected or not active.
		 * TRUE: Mode 4 is selected and active. */
		S_Mode4Sel : SAFEBOOL := FALSE;
		/* Indicates that mode 5 is selected and acknowledged.
		 * FALSE: Mode 5 is not selected or not active.
		 * TRUE: Mode 5 is selected and active. */
		S_Mode5Sel : SAFEBOOL := FALSE;
		/* Indicates that mode 6 is selected and acknowledged.
		 * FALSE: Mode 6 is not selected or not active.
		 * TRUE: Mode 6 is selected and active. */
		S_Mode6Sel : SAFEBOOL := FALSE;
		/* Indicates that mode 7 is selected and acknowledged.
		 * FALSE: Mode 7 is not selected or not active.
		 * TRUE: Mode 7 is selected and active. */
		S_Mode7Sel : SAFEBOOL := FALSE;
		/* Indicates that any of the 8 modes is selected and acknowledged.
		 * FALSE: No S_ModeX is selected.
		 * TRUE: One of the 8 S_ModeX is selected and active. */
		S_AnyModeSel : SAFEBOOL := FALSE;
		/* Optional. See 5.1.2 General Output Parameters */
		SafetyDemand : BOOL := FALSE;
		/* Optional. See 5.1.2 General Output Parameters */
		ResetRequest : BOOL := FALSE;
		/* See Section 5.1.2 General Output Parameters */
		Error : BOOL := FALSE;
		/* See Section 5.1.2 General Output Parameters */
		DiagCode : WORD := 16#0000;
	END_VAR

	VAR
		R_Trig_Reset : R_TRIG;
		R_Trig_S_SetMode : R_TRIG;

		ModeMonitorTimer : TON;
	END_VAR

	VAR_TEMP
		OneS_ModeChanged : BOOL;

		modeState : ModeState;
	END_VAR

	IF(NOT Activate) THEN
		DiagCode := TO_WORD(SF_ModeSelector_State#Idle);
		ModeMonitorTimer(IN := FALSE);
	ELSE

		modeState := DetermineModeState(S_Mode0, S_Mode1, S_Mode2, S_Mode3, S_Mode4, S_Mode5, S_Mode6, S_Mode7);

		ModeMonitorTimer(IN := modeState = ModeState#No_S_ModeX, PT := ModeMonitorTime);

		OneS_ModeChanged := S_Mode0 <> S_Mode0Sel OR S_Mode1 <> S_Mode1Sel OR S_Mode2 <> S_Mode2Sel OR S_Mode3 <> S_Mode3Sel OR S_Mode4 <> S_Mode4Sel OR S_Mode5 <> S_Mode5Sel OR S_Mode6 <> S_Mode6Sel OR S_Mode7 <> S_Mode7Sel;

		R_Trig_Reset(Reset);
		R_Trig_S_SetMode(IS(S_SetMode));

		CASE TO_UINT(DiagCode) OF
			SF_ModeSelector_State#Idle:
				/* IF(Activate) THEN - Active is always true here */
					DiagCode := TO_WORD(SF_ModeSelector_State#Mode_Changed);
			SF_ModeSelector_State#Mode_Changed:
				IF(modeState = ModeState#More_Than_One_S_ModeX) THEN
					DiagCode := TO_WORD(SF_ModeSelector_State#Error_Short_Circuit);
				ELSIF(ModeMonitorTimer.Q) THEN
					DiagCode := TO_WORD(SF_ModeSelector_State#Error_Open_Circuit);
				ELSIF((AutoSetMode OR R_Trig_S_SetMode.Q) AND IS(S_Unlock) AND modeState = ModeState#Only_One_S_ModeX) THEN
					DiagCode := TO_WORD(SF_ModeSelector_State#Mode_Selected);
				END_IF;
			SF_ModeSelector_State#Error_Short_Circuit, SF_ModeSelector_State#Error_Short_Circuit_Fixed:
				IF(Reset AND NOT R_Trig_Reset.Q) THEN
					DiagCode := TO_WORD(SF_ModeSelector_State#Reset_Error_1);
				ELSIF((modeState = ModeState#Only_One_S_ModeX OR modeState = ModeState#No_S_ModeX) AND R_Trig_Reset.Q) THEN
					DiagCode := TO_WORD(SF_ModeSelector_State#Mode_Changed);
				ELSE
					DiagCode := TO_WORD(DetermineErrorShortCircuit(modeState));
				END_IF;
			SF_ModeSelector_State#Error_Open_Circuit, SF_ModeSelector_State#Error_Open_Circuit_Fixed:
				IF(Reset AND NOT R_Trig_Reset.Q) THEN
					DiagCode := TO_WORD(SF_ModeSelector_State#Reset_Error_2);
				ELSIF(modeState = ModeState#Only_One_S_ModeX AND R_Trig_Reset.Q) THEN
					DiagCode := TO_WORD(SF_ModeSelector_State#Mode_Changed);
				ELSE
					DiagCode := TO_WORD(DetermineErrorOpenCircuit(modeState));
				END_IF;
			 SF_ModeSelector_State#Reset_Error_1:
				IF(NOT Reset) THEN
					DiagCode := TO_WORD(DetermineErrorShortCircuit(modeState));
				END_IF;
			SF_ModeSelector_State#Reset_Error_2:
				IF(NOT Reset) THEN
					DiagCode := TO_WORD(DetermineErrorOpenCircuit(modeState));
				END_IF;
			SF_ModeSelector_State#Mode_Selected:
				IF(modeState = ModeState#More_Than_One_S_ModeX) THEN
					DiagCode := TO_WORD(DetermineErrorShortCircuit(modeState));
				ELSIF(OneS_ModeChanged) THEN
					DiagCode := TO_WORD(SF_ModeSelector_State#Mode_Changed);
				ELSIF(IS_NOT(S_Unlock)) THEN
					DiagCode := TO_WORD(SF_ModeSelector_State#Mode_Locked);
				END_IF;
			SF_ModeSelector_State#Mode_Locked:
				IF(modeState = ModeState#More_Than_One_S_ModeX AND IS(S_Unlock)) THEN
					DiagCode := TO_WORD(DetermineErrorShortCircuit(modeState));
				ELSIF(OneS_ModeChanged AND IS(S_Unlock)) THEN
					DiagCode := TO_WORD(SF_ModeSelector_State#Mode_Changed);
				ELSIF(IS(S_Unlock)) THEN
					DiagCode := TO_WORD(SF_ModeSelector_State#Mode_Selected);
				END_IF;
		END_CASE;
	END_IF;

	CASE TO_UINT(DiagCode) OF
		SF_ModeSelector_State#Error_Short_Circuit_Fixed,
		SF_ModeSelector_State#Error_Open_Circuit_Fixed:
			Ready := TRUE;
			SafetyDemand := FALSE;
			ResetRequest := TRUE;
			Error := TRUE;
			S_AnyModeSel := SAFEBOOL_Constant#SAFEFALSE;
			S_Mode0Sel := SAFEBOOL_Constant#SAFEFALSE;
			S_Mode1Sel := SAFEBOOL_Constant#SAFEFALSE;
			S_Mode2Sel := SAFEBOOL_Constant#SAFEFALSE;
			S_Mode3Sel := SAFEBOOL_Constant#SAFEFALSE;
			S_Mode4Sel := SAFEBOOL_Constant#SAFEFALSE;
			S_Mode5Sel := SAFEBOOL_Constant#SAFEFALSE;
			S_Mode6Sel := SAFEBOOL_Constant#SAFEFALSE;
			S_Mode7Sel := SAFEBOOL_Constant#SAFEFALSE;
		SF_ModeSelector_State#Error_Short_Circuit,
		SF_ModeSelector_State#Error_Open_Circuit,
		SF_ModeSelector_State#Reset_Error_1,
		SF_ModeSelector_State#Reset_Error_2:
			Ready := TRUE;
			SafetyDemand := FALSE;
			ResetRequest := FALSE;
			Error := TRUE;
			S_AnyModeSel := SAFEBOOL_Constant#SAFEFALSE;
			S_Mode0Sel := SAFEBOOL_Constant#SAFEFALSE;
			S_Mode1Sel := SAFEBOOL_Constant#SAFEFALSE;
			S_Mode2Sel := SAFEBOOL_Constant#SAFEFALSE;
			S_Mode3Sel := SAFEBOOL_Constant#SAFEFALSE;
			S_Mode4Sel := SAFEBOOL_Constant#SAFEFALSE;
			S_Mode5Sel := SAFEBOOL_Constant#SAFEFALSE;
			S_Mode6Sel := SAFEBOOL_Constant#SAFEFALSE;
			S_Mode7Sel := SAFEBOOL_Constant#SAFEFALSE;
		SF_ModeSelector_State#Idle:
			Ready := FALSE;
			SafetyDemand := FALSE;
			ResetRequest := FALSE;
			Error := FALSE;
			S_AnyModeSel := SAFEBOOL_Constant#SAFEFALSE;
			S_Mode0Sel := SAFEBOOL_Constant#SAFEFALSE;
			S_Mode1Sel := SAFEBOOL_Constant#SAFEFALSE;
			S_Mode2Sel := SAFEBOOL_Constant#SAFEFALSE;
			S_Mode3Sel := SAFEBOOL_Constant#SAFEFALSE;
			S_Mode4Sel := SAFEBOOL_Constant#SAFEFALSE;
			S_Mode5Sel := SAFEBOOL_Constant#SAFEFALSE;
			S_Mode6Sel := SAFEBOOL_Constant#SAFEFALSE;
			S_Mode7Sel := SAFEBOOL_Constant#SAFEFALSE;
		SF_ModeSelector_State#Mode_Changed:
			Ready := TRUE;
			SafetyDemand := TRUE;
			ResetRequest := FALSE;
			Error := FALSE;
			S_AnyModeSel := SAFEBOOL_Constant#SAFEFALSE;
			S_Mode0Sel := SAFEBOOL_Constant#SAFEFALSE;
			S_Mode1Sel := SAFEBOOL_Constant#SAFEFALSE;
			S_Mode2Sel := SAFEBOOL_Constant#SAFEFALSE;
			S_Mode3Sel := SAFEBOOL_Constant#SAFEFALSE;
			S_Mode4Sel := SAFEBOOL_Constant#SAFEFALSE;
			S_Mode5Sel := SAFEBOOL_Constant#SAFEFALSE;
			S_Mode6Sel := SAFEBOOL_Constant#SAFEFALSE;
			S_Mode7Sel := SAFEBOOL_Constant#SAFEFALSE;
		SF_ModeSelector_State#Mode_Selected:
			Ready := TRUE;
			SafetyDemand := FALSE;
			ResetRequest := FALSE;
			Error := FALSE;
			S_AnyModeSel := SAFEBOOL_Constant#SAFETRUE;
			S_Mode0Sel := S_Mode0;
			S_Mode1Sel := S_Mode1;
			S_Mode2Sel := S_Mode2;
			S_Mode3Sel := S_Mode3;
			S_Mode4Sel := S_Mode4;
			S_Mode5Sel := S_Mode5;
			S_Mode6Sel := S_Mode6;
			S_Mode7Sel := S_Mode7;
		SF_ModeSelector_State#Mode_Locked:
			Ready := TRUE;
			SafetyDemand := FALSE;
			ResetRequest := FALSE;
			Error := FALSE;
			S_AnyModeSel := SAFEBOOL_Constant#SAFETRUE;
	END_CASE;

	ENO := ENO AND CheckSAFEBOOL(S_Mode0) AND CheckSAFEBOOL(S_Mode1) AND CheckSAFEBOOL(S_Mode2) AND CheckSAFEBOOL(S_Mode3) AND CheckSAFEBOOL(S_Mode4) AND CheckSAFEBOOL(S_Mode5) AND CheckSAFEBOOL(S_Mode6) AND CheckSAFEBOOL(S_Mode7) AND CheckSAFEBOOL(S_Unlock) AND CheckSAFEBOOL(S_SetMode);

END_FUNCTION_BLOCK

FUNCTION DetermineModeState : INT

	VAR_INPUT
		S_Mode0 : SAFEBOOL;
		S_Mode1 : SAFEBOOL;
		S_Mode2 : SAFEBOOL;
		S_Mode3 : SAFEBOOL;
		S_Mode4 : SAFEBOOL;
		S_Mode5 : SAFEBOOL;
		S_Mode6 : SAFEBOOL;
		S_Mode7 : SAFEBOOL;
	END_VAR

	IF(XOR(IS(S_Mode0),IS(S_Mode1),IS(S_Mode2),IS(S_Mode3),IS(S_Mode4),IS(S_Mode5),IS(S_Mode6),IS(S_Mode7))) THEN
		DetermineModeState := ModeState#Only_One_S_ModeX;
	ELSIF(NOT OR(IS(S_Mode0),IS(S_Mode1),IS(S_Mode2),IS(S_Mode3),IS(S_Mode4),IS(S_Mode5),IS(S_Mode6),IS(S_Mode7))) THEN
		DetermineModeState := ModeState#No_S_ModeX;
	ELSE
		DetermineModeState := ModeState#More_Than_One_S_ModeX;
	END_IF;
END_FUNCTION

FUNCTION DetermineErrorShortCircuit : UINT
	VAR_INPUT
		modeState : ModeState;
	END_VAR

	IF(modeState = ModeState#Only_One_S_ModeX OR modeState = ModeState#No_S_ModeX) THEN
		DetermineErrorShortCircuit := SF_ModeSelector_State#Error_Short_Circuit_Fixed;
	ELSE
		DetermineErrorShortCircuit := SF_ModeSelector_State#Error_Short_Circuit;
	END_IF;
END_FUNCTION

FUNCTION DetermineErrorOpenCircuit : UINT
	VAR_INPUT
		modeState : ModeState;
	END_VAR

	IF(modeState = ModeState#Only_One_S_ModeX) THEN
		DetermineErrorOpenCircuit := SF_ModeSelector_State#Error_Open_Circuit_Fixed;
	ELSE
		DetermineErrorOpenCircuit := SF_ModeSelector_State#Error_Open_Circuit;
	END_IF;
END_FUNCTION

END_NAMESPACE
END_NAMESPACE

(* ---- SF_MutingPar_2Sensor.iecst ---- *)
USING logicals.web.standard.safe;

NAMESPACE logicals.web.standard.safe
NAMESPACE plcopen

TYPE
	SF_MutingPar_2Sensor_State : UINT(
	/* Static Reset condition detected after FB activation in state 8401. */
	Reset_Error_1 := 16#C001,
	/* Static Reset condition detected in state 8402. */
	Reset_Error_2 := 16#C011,
	/* Error detected in muting sequence state 8000, 8010, 8310. */
	Error_Muting_Sequence_Base := 16#C004,
	/* DiscTimeEntry or MaxMutingTime value out of range. */
	Parameter_Error := 16#C010,
	/* Timing error: Active muting time (when S_MutingActive = TRUE) ex-ceeds MaxMutingTime. */
	Error_Timer_MaxMuting := 16#C020,
	/* Timing error: Discrepancy time for switching MutingSwitch11 and MutingSwitch12 from FALSE to TRUE > DiscTimeEntry. */
	Error_Timer_Entry := 16#C030,
	/* The function block is not active (initial state). */
	Idle := 16#0000,
	/* Muting not active and no safety demand from AOPD. If timers from subsequent muting are still running, they are stopped. */
	AOPD_Free := 16#8000,
	/* Function block was activated. */
	Init := 16#8401,
	/* Safety demand detected by AOPD, muting not active. */
	Safety_Demand_AOPD := 16#8802,
	/* Safety demand or errors have been detected and are now cleared. Operator acknowledgment by Reset required. */
	Wait_For_Reset := 16#8402,
	/* Safety function activated. */
	Safe := 16#8804,
	/* Muting sequence is in starting phase after rising trigger of MutingSwitch11. Monitoring of DiscTimeEntry is activated. */
	Muting_Start_1 := 16#8010,
	/* Muting sequence is in starting phase after rising trigger of MutingSwitch12. Monitoring of DiscTimeEntry is activated. */
	Muting_Start_2 := 16#8310,
	/* Muting sequence is active either:
	 * - After rising trigger of the second MutingSwitch 12 or 11 has been detected.
	 * - When both MutingSwitch 11 and 12 have been actuated in the same cycle.
	 * Monitoring of DiscTimeEntry is stopped. Monitoring of MaxMutingTime is activated.
	 */
	Muting_Active := 16#8020
	);
END_TYPE

/* Muting is the intended suppression of the safety function. In this FB, parallel muting with two muting sensors is specified. */
FUNCTION_BLOCK SF_MutingPar_2Sensor
	{ altName:="SF_MutingPar_2Sensor"; bgColor:="Gold"; width:=420; }
	VAR_INPUT
		/* See Section 5.1.1 General Input Parameters */
		Activate : BOOL := FALSE;
		/* Variable.
		 * OSSD signal from AOPD.
		 * FALSE: Protection field interrupted.
		 * TRUE: Protection field not interrupted. */
		S_AOPD_In : SAFEBOOL := SAFEBOOL_Constant#SAFEFALSE;
		/* Variable.
		 * Status of Muting sensor 11.
		 * FALSE: Muting sensor 11 not actuated.
		 * TRUE: Workpiece actuates muting sensor 11.
		 * Depending on the safety requirements it can be necessary to connect a SAFEBOOL. */
		MutingSwitch11 : BOOL := FALSE;
		/* Variable.
		 * Status of Muting sensor 12.
		 * FALSE: Muting sensor 12 not actuated.
		 * TRUE: Workpiece actuates muting sensor 12.
		 * Depending on the safety requirements it can be necessary to connect a SAFEBOOL. */
		MutingSwitch12 : BOOL := FALSE;
		/* Constant 0..4 s;
		 * Max. discrepancy time for S_MutingSwitch11 and S_MutingSwitch12 entering muting gate */
		DiscTimeEntry : TIME := T#0s;
		/* Constant 0..120 min;
		 * Maximum time for complete muting sequence, timer started when both muting sensors are actuated. */
		MaxMutingTime : TIME := T#0s;
		/* Variable or constant.
		 * Command by the control system that enables the start of the muting function when needed by the machine cycle. After the start of the muting function, this signal can be switched off.
		 * FALSE: Muting not enabled
		 * TRUE: Start of Muting function enabled */
		MutingEnable : BOOL := FALSE;
		/* See Section 5.1.1 General Input Parameters */
		S_StartReset : SAFEBOOL := SAFEBOOL_Constant#SAFEFALSE;
		/* See Section 5.1.1 General Input Parameters */
		Reset : BOOL := FALSE;
	END_VAR

	VAR_OUTPUT
		/* See Section 5.1.2 General Output Parameters */
		Ready : BOOL := FALSE;
		/* Safety related output, indicates status of the muted guard.
		 * FALSE: AOPD protection field interrupted and muting not active.
		 * TRUE: AOPD protection field not interrupted or muting active. */
		S_AOPD_Out : SAFEBOOL := SAFEBOOL_Constant#SAFEFALSE;
		/* Indicates status of Muting process.
		 * FALSE: Muting not active.
		 * TRUE: Muting active. */
		S_MutingActive : SAFEBOOL := SAFEBOOL_Constant#SAFEFALSE;
		/* Optional. See 5.1.2 General Output Parameters */
		SafetyDemand : BOOL := FALSE;
		/* Optional. See 5.1.2 General Output Parameters */
		ResetRequest : BOOL := FALSE;
		/* See Section 5.1.2 General Output Parameters */
		Error : BOOL := FALSE;
		/* See Section 5.1.2 General Output Parameters */
		DiagCode : WORD := 16#0000;
	END_VAR

	VAR
		/* ControlCode is used for state tracking */
		ControlCode : UINT := 16#0000;
		MutingTimer : TON;
		DiscTimeEntryTimer : TON;
		R_Trig_Reset : R_TRIG;
		R_Trig_S11 : R_TRIG;
		R_Trig_S12 : R_TRIG;
	END_VAR

	R_Trig_Reset(Reset);
	R_Trig_S11(MutingSwitch11);
	R_Trig_S12(MutingSwitch12);

	IF(NOT Activate) THEN
		ControlCode := SF_MutingPar_2Sensor_State#Idle;
		DiagCode := TO_WORD(ControlCode);
	ELSE
		CASE TO_UINT(ControlCode) OF
			SF_MutingPar_2Sensor_State#Idle:
				/* IF(Activate) THEN - Active is always true here */
					ControlCode := SF_MutingPar_2Sensor_State#Init;
					DiagCode := TO_WORD(ControlCode);
			SF_MutingPar_2Sensor_State#Init:
				IF(Reset AND NOT R_Trig_Reset.Q) THEN
					ControlCode := SF_MutingPar_2Sensor_State#Reset_Error_1;
					DiagCode := TO_WORD(ControlCode);
				ELSIF(DiscTimeEntry < T#0s OR DiscTimeEntry > T#4s OR MaxMutingTime < T#0s OR MaxMutingTime > T#120m) THEN
					ControlCode := SF_MutingPar_2Sensor_State#Parameter_Error;
					DiagCode := TO_WORD(ControlCode);
				ELSIF(R_Trig_Reset.Q OR IS(S_StartReset)) THEN
					ControlCode := SF_MutingPar_2Sensor_State#Safe;
					DiagCode := TO_WORD(ControlCode);
				END_IF;
			SF_MutingPar_2Sensor_State#Safe:
				IF(IS_NOT(S_AOPD_In)) THEN
					ControlCode := SF_MutingPar_2Sensor_State#Safety_Demand_AOPD;
					DiagCode := TO_WORD(ControlCode);
				ELSE
					ControlCode := SF_MutingPar_2Sensor_State#AOPD_Free;
					DiagCode := TO_WORD(ControlCode);
				END_IF;
			SF_MutingPar_2Sensor_State#Safety_Demand_AOPD:
				IF(IS(S_AOPD_In)) THEN
					ControlCode := SF_MutingPar_2Sensor_State#Wait_For_Reset;
					DiagCode := TO_WORD(ControlCode);
				END_IF;
			SF_MutingPar_2Sensor_State#Wait_For_Reset:
				IF(Reset AND NOT R_Trig_Reset.Q) THEN
					ControlCode := SF_MutingPar_2Sensor_State#Reset_Error_2;
					DiagCode := TO_WORD(ControlCode);
				ELSIF(R_Trig_Reset.Q) THEN
					ControlCode := SF_MutingPar_2Sensor_State#Safe;
					DiagCode := TO_WORD(ControlCode);
				END_IF;
			SF_MutingPar_2Sensor_State#AOPD_Free:
				IF((R_Trig_S11.Q AND MutingSwitch12 AND NOT R_Trig_S12.Q) OR
				   (R_Trig_S12.Q AND MutingSwitch11 AND NOT R_Trig_S11.Q) OR
				   ((MutingSwitch11 AND NOT R_Trig_S11.Q) AND (MutingSwitch12 AND NOT R_Trig_S12.Q)) OR
				   (NOT MutingEnable AND R_Trig_S11.Q) OR
				   (NOT MutingEnable AND R_Trig_S12.Q )) THEN
					ControlCode := SF_MutingPar_2Sensor_State#Error_Muting_Sequence_Base;
					IF(MutingEnable) THEN
						DiagCode := TO_WORD(SF_MutingPar_2Sensor_State#Error_Muting_Sequence_Base + GetErrorStateOfMutingSensors(MutingSwitch11, MutingSwitch12));
					ELSE
						DiagCode := TO_WORD(SF_MutingPar_2Sensor_State#Error_Muting_Sequence_Base + 16#0F00 + GetErrorStateOfMutingSensors(MutingSwitch11, MutingSwitch12));
					END_IF;
				ELSIF(IS_NOT(S_AOPD_In)) THEN
					ControlCode := SF_MutingPar_2Sensor_State#Safety_Demand_AOPD;
					DiagCode := TO_WORD(ControlCode);
				ELSIF(MutingEnable AND R_Trig_S11.Q AND NOT MutingSwitch12) THEN
					ControlCode := SF_MutingPar_2Sensor_State#Muting_Start_1;
					DiagCode := TO_WORD(ControlCode);
				ELSIF(MutingEnable AND NOT MutingSwitch11 AND R_Trig_S12.Q) THEN
					ControlCode := SF_MutingPar_2Sensor_State#Muting_Start_2;
					DiagCode := TO_WORD(ControlCode);
				ELSIF(MutingEnable AND R_Trig_S11.Q AND R_Trig_S12.Q) THEN
					ControlCode := SF_MutingPar_2Sensor_State#Muting_Active;
					DiagCode := TO_WORD(ControlCode);
				END_IF;
			SF_MutingPar_2Sensor_State#Muting_Start_1:
				MutingTimer();
				DiscTimeEntryTimer();

				IF(NOT MutingEnable OR NOT MutingSwitch11) THEN
					ControlCode := SF_MutingPar_2Sensor_State#Error_Muting_Sequence_Base;
					IF(MutingEnable) THEN
						DiagCode := TO_WORD(SF_MutingPar_2Sensor_State#Error_Muting_Sequence_Base + 16#0100 + GetErrorStateOfMutingSensors(MutingSwitch11, MutingSwitch12));
					ELSE
						DiagCode := TO_WORD(SF_MutingPar_2Sensor_State#Error_Muting_Sequence_Base + 16#0F00 + GetErrorStateOfMutingSensors(MutingSwitch11, MutingSwitch12));
					END_IF;
				ELSIF(MutingTimer.Q) THEN
					ControlCode := SF_MutingPar_2Sensor_State#Error_Timer_MaxMuting;
					DiagCode := TO_WORD(ControlCode);
				ELSIF(DiscTimeEntryTimer.Q) THEN
					ControlCode := SF_MutingPar_2Sensor_State#Error_Timer_Entry;
					DiagCode := TO_WORD(ControlCode);
				ELSIF(IS_NOT(S_AOPD_In)) THEN
					ControlCode := SF_MutingPar_2Sensor_State#Safety_Demand_AOPD;
					DiagCode := TO_WORD(ControlCode);
				ELSIF(MutingEnable AND MutingSwitch11 AND R_Trig_S12.Q) THEN
					ControlCode := SF_MutingPar_2Sensor_State#Muting_Active;
					DiagCode := TO_WORD(ControlCode);
				END_IF;
			SF_MutingPar_2Sensor_State#Muting_Start_2:
				MutingTimer();
				DiscTimeEntryTimer();

				IF(NOT MutingEnable OR NOT MutingSwitch12) THEN
					ControlCode := SF_MutingPar_2Sensor_State#Error_Muting_Sequence_Base;
					IF(MutingEnable) THEN
						DiagCode := TO_WORD(SF_MutingPar_2Sensor_State#Error_Muting_Sequence_Base + 16#0200 + GetErrorStateOfMutingSensors(MutingSwitch11, MutingSwitch12));
					ELSE
						DiagCode := TO_WORD(SF_MutingPar_2Sensor_State#Error_Muting_Sequence_Base + 16#0F00 + GetErrorStateOfMutingSensors(MutingSwitch11, MutingSwitch12));
					END_IF;
				ELSIF(MutingTimer.Q) THEN
					ControlCode := SF_MutingPar_2Sensor_State#Error_Timer_MaxMuting;
					DiagCode := TO_WORD(ControlCode);
				ELSIF(DiscTimeEntryTimer.Q) THEN
					ControlCode := SF_MutingPar_2Sensor_State#Error_Timer_Entry;
					DiagCode := TO_WORD(ControlCode);
				ELSIF(IS_NOT(S_AOPD_In)) THEN
					ControlCode := SF_MutingPar_2Sensor_State#Safety_Demand_AOPD;
					DiagCode := TO_WORD(ControlCode);
				ELSIF(MutingEnable AND R_Trig_S11.Q AND MutingSwitch12) THEN
					ControlCode := SF_MutingPar_2Sensor_State#Muting_Active;
					DiagCode := TO_WORD(ControlCode);
				END_IF;
			SF_MutingPar_2Sensor_State#Muting_Active:
				MutingTimer();
				DiscTimeEntryTimer();

				IF(MutingTimer.Q) THEN
					ControlCode := SF_MutingPar_2Sensor_State#Error_Timer_MaxMuting;
					DiagCode := TO_WORD(ControlCode);
				ELSIF(NOT MutingSwitch11 OR NOT MutingSwitch12) THEN
					ControlCode := SF_MutingPar_2Sensor_State#AOPD_Free;
					DiagCode := TO_WORD(ControlCode);
				END_IF;
			SF_MutingPar_2Sensor_State#Error_Muting_Sequence_Base:
				IF(NOT (MutingSwitch11 OR MutingSwitch12)) THEN
					ControlCode := SF_MutingPar_2Sensor_State#Wait_For_Reset;
					DiagCode := TO_WORD(ControlCode);
				END_IF;
			SF_MutingPar_2Sensor_State#Error_Timer_MaxMuting,
			SF_MutingPar_2Sensor_State#Error_Timer_Entry:
				IF(NOT (MutingSwitch11 OR MutingSwitch12)) THEN
					ControlCode := SF_MutingPar_2Sensor_State#Wait_For_Reset;
					DiagCode := TO_WORD(ControlCode);
				END_IF;
			SF_MutingPar_2Sensor_State#Reset_Error_1:
				IF(NOT Reset) THEN
					ControlCode := SF_MutingPar_2Sensor_State#Init;
					DiagCode := TO_WORD(ControlCode);
				END_IF;
			SF_MutingPar_2Sensor_State#Reset_Error_2:
				IF(NOT Reset) THEN
					ControlCode := SF_MutingPar_2Sensor_State#Wait_For_Reset;
					DiagCode := TO_WORD(ControlCode);
				END_IF;
		END_CASE;
	END_IF;

	CASE TO_UINT(ControlCode) OF
		SF_MutingPar_2Sensor_State#Idle:
			DiscTimeEntryTimer(IN := FALSE);
			MutingTimer(IN := FALSE);
			Ready := FALSE;
			S_AOPD_Out := SAFEBOOL_Constant#SAFEFALSE;
			S_MutingActive := SAFEBOOL_Constant#SAFEFALSE;
			SafetyDemand := FALSE;
			ResetRequest := FALSE;
			Error := FALSE;
		SF_MutingPar_2Sensor_State#AOPD_Free:
			DiscTimeEntryTimer(IN := FALSE);
			MutingTimer(IN := FALSE);
			Ready := TRUE;
			S_AOPD_Out := SAFEBOOL_Constant#SAFETRUE;
			S_MutingActive := SAFEBOOL_Constant#SAFEFALSE;
			SafetyDemand := FALSE;
			ResetRequest := FALSE;
			Error := FALSE;
		SF_MutingPar_2Sensor_State#Init,
		SF_MutingPar_2Sensor_State#Wait_For_Reset:
			DiscTimeEntryTimer(IN := FALSE);
			MutingTimer(IN := FALSE);
			Ready := TRUE;
			S_AOPD_Out := SAFEBOOL_Constant#SAFEFALSE;
			S_MutingActive := SAFEBOOL_Constant#SAFEFALSE;
			SafetyDemand := FALSE;
			ResetRequest := TRUE;
			Error := FALSE;
		SF_MutingPar_2Sensor_State#Safety_Demand_AOPD:
			DiscTimeEntryTimer(IN := FALSE);
			MutingTimer(IN := FALSE);
			Ready := TRUE;
			S_AOPD_Out := SAFEBOOL_Constant#SAFEFALSE;
			S_MutingActive := SAFEBOOL_Constant#SAFEFALSE;
			SafetyDemand := TRUE;
			ResetRequest := FALSE;
			Error := FALSE;
		SF_MutingPar_2Sensor_State#Safe:
			DiscTimeEntryTimer(IN := FALSE);
			MutingTimer(IN := FALSE);
			Ready := TRUE;
			S_AOPD_Out := SAFEBOOL_Constant#SAFEFALSE;
			S_MutingActive := SAFEBOOL_Constant#SAFEFALSE;
			SafetyDemand := FALSE;
			ResetRequest := FALSE;
			Error := FALSE;
		SF_MutingPar_2Sensor_State#Muting_Start_1,
		SF_MutingPar_2Sensor_State#Muting_Start_2:
			DiscTimeEntryTimer(IN := TRUE, PT := DiscTimeEntry);
			MutingTimer(IN := TRUE, PT := MaxMutingTime);
			Ready := TRUE;
			S_AOPD_Out := SAFEBOOL_Constant#SAFETRUE;
			S_MutingActive := SAFEBOOL_Constant#SAFEFALSE;
			SafetyDemand := FALSE;
			ResetRequest := FALSE;
			Error := FALSE;
		SF_MutingPar_2Sensor_State#Muting_Active:
			DiscTimeEntryTimer(IN := FALSE);
			MutingTimer(IN := TRUE, PT := MaxMutingTime);
			Ready := TRUE;
			S_AOPD_Out := SAFEBOOL_Constant#SAFETRUE;
			S_MutingActive := SAFEBOOL_Constant#SAFETRUE;
			SafetyDemand := FALSE;
			ResetRequest := FALSE;
			Error := FALSE;
		SF_MutingPar_2Sensor_State#Reset_Error_1,
		SF_MutingPar_2Sensor_State#Reset_Error_2,
		SF_MutingPar_2Sensor_State#Error_Muting_Sequence_Base,
		SF_MutingPar_2Sensor_State#Parameter_Error,
		SF_MutingPar_2Sensor_State#Error_Timer_MaxMuting,
		SF_MutingPar_2Sensor_State#Error_Timer_Entry:
			DiscTimeEntryTimer(IN := FALSE);
			MutingTimer(IN := FALSE);
			Ready := TRUE;
			S_AOPD_Out := SAFEBOOL_Constant#SAFEFALSE;
			S_MutingActive := SAFEBOOL_Constant#SAFEFALSE;
			SafetyDemand := FALSE;
			ResetRequest := FALSE;
			Error := TRUE;
	END_CASE;

	ENO := ENO AND CheckSAFEBOOL(S_AOPD_In) AND CheckSAFEBOOL(S_StartReset);

END_FUNCTION_BLOCK

/* returns a UINT that can be added to the DiagCode indicating which muting states were active prior to the Error */
FUNCTION GetErrorStateOfMutingSensors : UINT
	VAR_INPUT
		MS_11 : BOOL;
		MS_12 : BOOL;
	END_VAR
	VAR
		Result : UINT := 16#0000;
	END_VAR

	IF(MS_11) THEN
		Result := Result + 16#0010;
	END_IF;
	IF(MS_12) THEN
		Result := Result + 16#0020;
	END_IF;

	GetErrorStateOfMutingSensors := Result;
END_FUNCTION

END_NAMESPACE
END_NAMESPACE

(* ---- SF_MutingSeq.iecst ---- *)
USING logicals.web.standard.safe;

NAMESPACE logicals.web.standard.safe
NAMESPACE plcopen

TYPE
	SF_MutingSeq_State : UINT(
	/* Static Reset condition detected after FB activation. */
	Reset_Error_1 := 16#C001,
	/* Static Reset condition detected in state 8402 */
	Reset_Error_2 := 16#C011,
	/* Error detected in muting sequence in states 8000, 8010, 8020, 8120 or 8110 */
	Error_Muting_Sequence_Base := 16#C004,
	/* MaxMutingTime value out of range */
	Parameter_Error := 16#C010,
	/* Error Timer MaxMuting */
	Error_Timer_MaxMuting := 16#C020,
	/* The function block is not active (initial state). */
	Idle := 16#0000,
	/* Muting not active and no safety demand from AOPD */
	AOPD_Free := 16#8000,
	/* Function block has been activated */
	Init := 16#8401,
	/* Safety demand detected by AOPD, muting not active */
	Safety_Demand_AOPD := 16#8802,
	/* Safety demand or errors have been detected and are now cleared. Operator acknowledgment by Reset required */
	Wait_for_Reset := 16#8402,
	/* Safety function activated */
	Safe := 16#8002,
	/* Muting forward, sequence is in starting phase and no safety demand */
	Muting_Forward_Start := 16#8010,
	/* Muting forward, sequence is active */
	Muting_Forward_Active := 16#8020,
	/* Muting Backward Active */
	Muting_Backward_Active := 16#8120,
	/* Muting Backward Start */
	Muting_Backward_Start := 16#8110);
END_TYPE

/*
 * Muting is the intended suppression of the safety function (e.g., light barriers). In this FB, sequential muting with four
 * muting sensors is specified.
 */
FUNCTION_BLOCK SF_MutingSeq
	{ altName:="SF_MutingSeq"; bgColor:="Gold"; width:=380; }
	VAR_INPUT
		/* See Section 5.1.1 General Input Parameters */
		Activate : BOOL := FALSE;
		/* Variable. OSSD signal from AOPD.
		 * FALSE: Protection field interrupted.
		 * TRUE: Protection field not interrupted. */
		S_AOPD_In : SAFEBOOL := SAFEBOOL_Constant#SAFEFALSE;
		/* Variable. Status of Muting sensor 11.
		 * FALSE: Muting sensor 11 not actuated.
		 * TRUE: Workpiece actuates muting sensor 11.
		 * Depending on the safety requirements it can be necessary to connect a SAFEBOOL. */
		MutingSwitch11 : BOOL := FALSE;
		/* Variable. Status of Muting sensor 12.
		 * FALSE: Muting sensor 12 not actuated.
		 * TRUE: Workpiece actuates muting sensor 12.
		 * Depending on the safety requirements it can be necessary to connect a SAFEBOOL. */
		MutingSwitch12 : BOOL := FALSE;
		/* Variable. Status of Muting sensor 21.
		 * FALSE: Muting sensor 21 not actuated.
		 * TRUE: Workpiece actuates muting sensor 21.
		 * Depending on the safety requirements it can be necessary to connect a SAFEBOOL. */
		MutingSwitch21 : BOOL := FALSE;
		/* Variable. Status of Muting sensor 22.
		 * FALSE: Muting sensor 22 not actuated.
		 * TRUE: Workpiece actuates muting sensor 22.
		 * Depending on the safety requirements it can be necessary to connect a SAFEBOOL. */
		MutingSwitch22 : BOOL := FALSE;
		/* Constant 0 .. 120 min (application specific).
		 * Maximum time for complete muting sequence, timer
		 * started when second muting sensor is actuated.
		 * If needed this can be combined with SF_Override. */
		MaxMutingTime : TIME := T#0s;
		/* Variable or constant. Command by the control system that enables the start of the
		 * muting function when needed by the machine cycle. After the start of the muting
		 * function, this signal can be switched off.
		 * FALSE: Muting not enabled
		 * TRUE: Start of Muting function enabled */
		MutingEnable : BOOL := FALSE;
		/* See Section 5.1.1 General Input Parameters */
		S_StartReset : SAFEBOOL := SAFEBOOL_Constant#SAFEFALSE;
		/* See Section 5.1.1 General Input Parameters */
		Reset : BOOL := FALSE;
	END_VAR
	VAR_OUTPUT
		/* See Section 5.1.2 General Output Parameters */
		Ready : BOOL := FALSE;
		/* Safety related output, indicates status of the muted guard.
		 * FALSE: AOPD protection field interrupted and muting not active.
		 * TRUE: AOPD protection field not interrupted or muting active. */
		S_AOPD_OUT : SAFEBOOL := SAFEBOOL_Constant#SAFEFALSE;
		/* Indicates status of Muting process.
		 * FALSE: Muting not active.
		 * TRUE: Muting active. */
		S_MutingActive : SAFEBOOL := SAFEBOOL_Constant#SAFEFALSE;
		/* Optional. See Section 5.1.2 General Output Parameters */
		SafetyDemand : BOOL := FALSE;
		/* Optional. See Section 5.1.2 General Output Parameters */
		ResetRequest : BOOL := FALSE;
		/* See Section 5.1.2 General Output Parameters */
		Error : BOOL := FALSE;
		/* See Section 5.1.2 General Output Parameters */
		DiagCode : WORD := 16#0000;
	END_VAR
	VAR
		/* ControlCode is used for state tracking */
		MutingTimer : TON;
		ControlCode : UINT := 16#0000;
		/* MutingSwitchState is used to produce the correct DiagCode for errors in the muting sequence in multiple states */
		MutingSwitchState : UINT := 16#0000;
		R_Trig_Reset : R_TRIG;
		R_Trig_S11 : R_TRIG;
		R_Trig_S12 : R_TRIG;
		R_Trig_S21 : R_TRIG;
		R_Trig_S22 : R_TRIG;
		F_Trig_S11 : F_TRIG;
		F_Trig_S12 : F_TRIG;
		F_Trig_S21 : F_TRIG;
		F_Trig_S22 : F_TRIG;
	END_VAR

	R_Trig_Reset(Reset);
	R_Trig_S11(MutingSwitch11);
	R_Trig_S12(MutingSwitch12);
	R_Trig_S21(MutingSwitch21);
	R_Trig_S22(MutingSwitch22);
	F_Trig_S11(MutingSwitch11);
	F_Trig_S12(MutingSwitch12);
	F_Trig_S21(MutingSwitch21);
	F_Trig_S22(MutingSwitch22);

	IF(NOT Activate) THEN
		ControlCode := SF_MutingSeq_State#Idle;
		DiagCode := TO_WORD(ControlCode);
	ELSE
		CASE TO_UINT(ControlCode) OF
			SF_MutingSeq_State#Idle:
				ControlCode := SF_MutingSeq_State#Init;
				DiagCode := TO_WORD(ControlCode);
			SF_MutingSeq_State#Init:
				IF(Reset AND NOT R_Trig_Reset.Q) THEN
					ControlCode := SF_MutingSeq_State#Reset_Error_1;
					DiagCode := TO_WORD(ControlCode);
				ELSIF(MaxMutingTime < T#0M OR MaxMutingTime > T#120M) THEN
					ControlCode := SF_MutingSeq_State#Parameter_Error;
					DiagCode := TO_WORD(ControlCode);
				ELSIF(R_Trig_Reset.Q OR IS(S_StartReset)) THEN
					ControlCode := SF_MutingSeq_State#Safe;
					DiagCode := TO_WORD(ControlCode);
				END_IF;
			SF_MutingSeq_State#Reset_Error_1:
				IF(NOT Reset) THEN
					ControlCode := SF_MutingSeq_State#Init;
					DiagCode := TO_WORD(ControlCode);
				END_IF;
			SF_MutingSeq_State#Safe:
				IF(IS_NOT(S_AOPD_In)) THEN
					ControlCode := SF_MutingSeq_State#Safety_Demand_AOPD;
					DiagCode := TO_WORD(ControlCode);
				ELSE
					ControlCode := SF_MutingSeq_State#AOPD_Free;
					DiagCode := TO_WORD(ControlCode);
				END_IF;
			SF_MutingSeq_State#Safety_Demand_AOPD:
				IF(IS(S_AOPD_In)) THEN
					ControlCode := SF_MutingSeq_State#Wait_for_Reset;
					DiagCode := TO_WORD(ControlCode);
				END_IF;
			SF_MutingSeq_State#Wait_for_Reset:
				IF(Reset AND NOT R_Trig_Reset.Q) THEN
					ControlCode := SF_MutingSeq_State#Reset_Error_2;
					DiagCode := TO_WORD(ControlCode);
				ELSIF(R_Trig_Reset.Q) THEN
					ControlCode := SF_MutingSeq_State#Safe;
					DiagCode := TO_WORD(ControlCode);
				END_IF;
			SF_MutingSeq_State#Reset_Error_2:
				IF(NOT Reset) THEN
					ControlCode := SF_MutingSeq_State#Wait_for_Reset;
					DiagCode := TO_WORD(ControlCode);
				END_IF;
			SF_MutingSeq_State#Error_Muting_Sequence_Base:
				IF(NOT (MutingSwitch11 OR MutingSwitch12 OR MutingSwitch21 OR MutingSwitch22)) THEN
					ControlCode := SF_MutingSeq_State#Wait_for_Reset;
					DiagCode := TO_WORD(ControlCode);
				END_IF;
			SF_MutingSeq_State#Error_Timer_MaxMuting:
				IF(NOT (MutingSwitch11 OR MutingSwitch12 OR MutingSwitch21 OR MutingSwitch22)) THEN
					ControlCode := SF_MutingSeq_State#Wait_for_Reset;
					DiagCode := TO_WORD(ControlCode);
				END_IF;
			SF_MutingSeq_State#AOPD_Free:
				IF((NOT MutingEnable AND R_Trig_S11.Q) OR (NOT MutingEnable AND R_Trig_S22.Q)) THEN
					/* Error muting sequence */
					ControlCode := SF_MutingSeq_State#Error_Muting_Sequence_Base;
					DiagCode := TO_WORD(SF_MutingSeq_State#Error_Muting_Sequence_Base + 16#0F00 + MutingSeqGetErrorStateOfMutingSensors(MutingSwitch11, MutingSwitch12, MutingSwitch21, MutingSwitch22));
				ELSIF((MutingSwitch12 OR MutingSwitch21) OR (MutingSwitch11 AND MutingSwitch22)) THEN
					/* Error muting sequence */
					ControlCode := SF_MutingSeq_State#Error_Muting_Sequence_Base;
					DiagCode := TO_WORD(SF_MutingSeq_State#Error_Muting_Sequence_Base + MutingSeqGetErrorStateOfMutingSensors(MutingSwitch11, MutingSwitch12, MutingSwitch21, MutingSwitch22));
				ELSIF(IS_NOT(S_AOPD_In)) THEN
					ControlCode := SF_MutingSeq_State#Safety_Demand_AOPD;
					DiagCode := TO_WORD(ControlCode);
				ELSIF(MutingEnable AND (R_Trig_S11.Q AND NOT MutingSwitch12 AND NOT MutingSwitch21 AND NOT MutingSwitch22)) THEN
					ControlCode := SF_MutingSeq_State#Muting_Forward_Start;
					DiagCode := TO_WORD(ControlCode);
				ELSIF(MutingEnable AND (NOT MutingSwitch11 AND NOT MutingSwitch12 AND NOT MutingSwitch21 AND R_Trig_S22.Q)) THEN
					ControlCode := SF_MutingSeq_State#Muting_Backward_Start;
					DiagCode := TO_WORD(ControlCode);
				END_IF;
			SF_MutingSeq_State#Muting_Forward_Start:
				IF(NOT MutingEnable) THEN
					/* Error muting sequence */
					ControlCode := SF_MutingSeq_State#Error_Muting_Sequence_Base;
					DiagCode := TO_WORD(SF_MutingSeq_State#Error_Muting_Sequence_Base + 16#0F00 + MutingSeqGetErrorStateOfMutingSensors(MutingSwitch11, MutingSwitch12, MutingSwitch21, MutingSwitch22));
				ELSIF(NOT MutingSwitch11 OR MutingSwitch21 OR MutingSwitch22) THEN
					/* Error muting sequence */
					ControlCode := SF_MutingSeq_State#Error_Muting_Sequence_Base;
					DiagCode := TO_WORD(SF_MutingSeq_State#Error_Muting_Sequence_Base + 16#0100 + MutingSeqGetErrorStateOfMutingSensors(MutingSwitch11, MutingSwitch12, MutingSwitch21, MutingSwitch22));
				ELSIF(IS_NOT(S_AOPD_In)) THEN
					ControlCode := SF_MutingSeq_State#Safety_Demand_AOPD;
					DiagCode := TO_WORD(ControlCode);
				ELSIF(MutingEnable AND MutingSwitch11 AND R_Trig_S12.Q AND NOT MutingSwitch21 AND NOT MutingSwitch22) THEN
					ControlCode := SF_MutingSeq_State#Muting_Forward_Active;
					DiagCode := TO_WORD(ControlCode);
				END_IF;
			SF_MutingSeq_State#Muting_Forward_Active:
				IF(NOT MutingEnable) THEN
					/* Error muting sequence */
					ControlCode := SF_MutingSeq_State#Error_Muting_Sequence_Base;
					DiagCode := TO_WORD(SF_MutingSeq_State#Error_Muting_Sequence_Base + 16#0F00 + MutingSeqGetErrorStateOfMutingSensors(MutingSwitch11, MutingSwitch12, MutingSwitch21, MutingSwitch22));
				ELSIF((R_Trig_S11.Q OR R_Trig_S12.Q OR F_Trig_S22.Q)
					OR(MutingSwitch11 AND F_Trig_S12.Q)
					OR((MutingSwitch11 OR MutingSwitch12) AND (F_Trig_S21.Q))
					OR((NOT MutingSwitch11 OR NOT MutingSwitch12) AND NOT MutingSwitch22)
					OR(((NOT MutingSwitch11 OR NOT MutingSwitch12) OR NOT MutingSwitch21) AND R_Trig_S22.Q)
					OR(R_Trig_S21.Q AND R_Trig_S22.Q)
					OR(F_Trig_S11.Q AND F_Trig_S12.Q)
					OR(F_Trig_S12.Q AND F_Trig_S21.Q)) THEN
					/* Error muting sequence */
					ControlCode := SF_MutingSeq_State#Error_Muting_Sequence_Base;
					DiagCode := TO_WORD(SF_MutingSeq_State#Error_Muting_Sequence_Base + 16#0200 + MutingSeqGetErrorStateOfMutingSensors(MutingSwitch11, MutingSwitch12, MutingSwitch21, MutingSwitch22));
				ELSIF(MutingTimer.Q) THEN
					ControlCode := SF_MutingSeq_State#Error_Timer_MaxMuting;
					DiagCode := TO_WORD(ControlCode);
				ELSIF(NOT MutingSwitch11 AND NOT MutingSwitch12 AND F_Trig_S21.Q AND MutingSwitch22) THEN
					ControlCode := SF_MutingSeq_State#AOPD_Free;
					DiagCode := TO_WORD(ControlCode);
				END_IF;
			SF_MutingSeq_State#Muting_Backward_Start:
				IF(NOT MutingEnable) THEN
					/* Error muting sequence */
					ControlCode := SF_MutingSeq_State#Error_Muting_Sequence_Base;
					DiagCode := TO_WORD(SF_MutingSeq_State#Error_Muting_Sequence_Base + 16#0F00 + MutingSeqGetErrorStateOfMutingSensors(MutingSwitch11, MutingSwitch12, MutingSwitch21, MutingSwitch22));
				ELSIF(MutingSwitch11 OR MutingSwitch12 OR NOT MutingSwitch22) THEN
					/* Error muting sequence */
					ControlCode := SF_MutingSeq_State#Error_Muting_Sequence_Base;
					DiagCode := TO_WORD(SF_MutingSeq_State#Error_Muting_Sequence_Base + 16#0300 + MutingSeqGetErrorStateOfMutingSensors(MutingSwitch11, MutingSwitch12, MutingSwitch21, MutingSwitch22));
				ELSIF(IS_NOT(S_AOPD_In)) THEN
					ControlCode := SF_MutingSeq_State#Safety_Demand_AOPD;
					DiagCode := TO_WORD(ControlCode);
				ELSIF(MutingEnable AND (NOT MutingSwitch11 AND NOT MutingSwitch12 AND R_Trig_S21.Q AND MutingSwitch22)) THEN
					ControlCode := SF_MutingSeq_State#Muting_Backward_Active;
					DiagCode := TO_WORD(ControlCode);
				END_IF;
			SF_MutingSeq_State#Muting_Backward_Active:
				IF(NOT MutingEnable) THEN
					/* Error muting sequence */
					ControlCode := SF_MutingSeq_State#Error_Muting_Sequence_Base;
					DiagCode := TO_WORD(SF_MutingSeq_State#Error_Muting_Sequence_Base + 16#0F00 + MutingSeqGetErrorStateOfMutingSensors(MutingSwitch11, MutingSwitch12, MutingSwitch21, MutingSwitch22));
				ELSIF((F_Trig_S11.Q OR R_Trig_S21.Q OR R_Trig_S22.Q)
					OR(MutingSwitch22 AND F_Trig_S21.Q)
					OR((MutingSwitch22 OR MutingSwitch21) AND F_Trig_S12.Q)
					OR((NOT MutingSwitch22 OR NOT MutingSwitch21) AND NOT MutingSwitch11)
					OR((NOT MutingSwitch22 OR NOT MutingSwitch21 OR NOT MutingSwitch12) AND R_Trig_S11.Q)
					OR(R_Trig_S11.Q AND R_Trig_S12.Q)
					OR(F_Trig_S22.Q AND F_Trig_S21.Q)
					OR(F_Trig_S21.Q AND F_Trig_S12.Q)) THEN
					/* Error muting sequence */
					ControlCode := SF_MutingSeq_State#Error_Muting_Sequence_Base;
					DiagCode := TO_WORD(SF_MutingSeq_State#Error_Muting_Sequence_Base + 16#0400 + MutingSeqGetErrorStateOfMutingSensors(MutingSwitch11, MutingSwitch12, MutingSwitch21, MutingSwitch22));
				ELSIF(MutingTimer.Q) THEN
					ControlCode := SF_MutingSeq_State#Error_Timer_MaxMuting;
					DiagCode := TO_WORD(ControlCode);
				ELSIF(MutingSwitch11 AND F_Trig_S12.Q AND NOT MutingSwitch21 AND NOT MutingSwitch22) THEN
					ControlCode := SF_MutingSeq_State#AOPD_Free;
					DiagCode := TO_WORD(ControlCode);
				END_IF;
		ELSE
			/* TODO evaluation of Parameter Error C010 ends here, is this intended? */
			ENO := FALSE;
		END_CASE;
	END_IF;

	CASE TO_UINT(ControlCode) OF
		SF_MutingSeq_State#Idle:
			MutingTimer(IN := FALSE);
			Ready := FALSE;
			S_AOPD_OUT := SAFEBOOL_Constant#SAFEFALSE;
			S_MutingActive := SAFEBOOL_Constant#SAFEFALSE;
			SafetyDemand := FALSE;
			ResetRequest := FALSE;
			Error := FALSE;
		SF_MutingSeq_State#Init:
			MutingTimer(IN := FALSE);
			Ready := TRUE;
			S_AOPD_OUT := SAFEBOOL_Constant#SAFEFALSE;
			S_MutingActive := SAFEBOOL_Constant#SAFEFALSE;
			SafetyDemand := FALSE;
			ResetRequest := TRUE;
			Error := FALSE;
		SF_MutingSeq_State#Reset_Error_1,
		SF_MutingSeq_State#Reset_Error_2,
		SF_MutingSeq_State#Error_Muting_Sequence_Base,
		SF_MutingSeq_State#Parameter_Error,
		SF_MutingSeq_State#Error_Timer_MaxMuting:
			MutingTimer(IN := FALSE);
			Ready := TRUE;
			S_AOPD_OUT := SAFEBOOL_Constant#SAFEFALSE;
			S_MutingActive := SAFEBOOL_Constant#SAFEFALSE;
			SafetyDemand := FALSE;
			ResetRequest := FALSE;
			Error := TRUE;
		SF_MutingSeq_State#AOPD_Free:
			MutingTimer(IN := FALSE);
			Ready := TRUE;
			S_AOPD_OUT := SAFEBOOL_Constant#SAFETRUE;
			S_MutingActive := SAFEBOOL_Constant#SAFEFALSE;
			SafetyDemand := FALSE;
			ResetRequest := FALSE;
			Error := FALSE;
		SF_MutingSeq_State#Safety_Demand_AOPD:
			MutingTimer(IN := FALSE);
			Ready := TRUE;
			S_AOPD_OUT := SAFEBOOL_Constant#SAFEFALSE;
			S_MutingActive := SAFEBOOL_Constant#SAFEFALSE;
			SafetyDemand := TRUE;
			ResetRequest := FALSE;
			Error := FALSE;
		SF_MutingSeq_State#Wait_for_Reset:
			MutingTimer(IN := FALSE);
			Ready := TRUE;
			S_AOPD_OUT := SAFEBOOL_Constant#SAFEFALSE;
			S_MutingActive := SAFEBOOL_Constant#SAFEFALSE;
			SafetyDemand := FALSE;
			ResetRequest := TRUE;
			Error := FALSE;
		SF_MutingSeq_State#Safe:
			MutingTimer(IN := FALSE);
			Ready := TRUE;
			S_AOPD_OUT := SAFEBOOL_Constant#SAFEFALSE;
			S_MutingActive := SAFEBOOL_Constant#SAFEFALSE;
			SafetyDemand := FALSE;
			ResetRequest := FALSE;
			Error := FALSE;
		SF_MutingSeq_State#Muting_Forward_Start:
			MutingTimer(IN := FALSE);
			Ready := TRUE;
			S_AOPD_OUT := SAFEBOOL_Constant#SAFETRUE;
			S_MutingActive := SAFEBOOL_Constant#SAFEFALSE;
			SafetyDemand := FALSE;
			ResetRequest := FALSE;
			Error := FALSE;
		SF_MutingSeq_State#Muting_Forward_Active:
			MutingTimer(IN := TRUE, PT := MaxMutingTime);
			Ready := TRUE;
			S_AOPD_OUT := SAFEBOOL_Constant#SAFETRUE;
			S_MutingActive := SAFEBOOL_Constant#SAFETRUE;
			SafetyDemand := FALSE;
			ResetRequest := FALSE;
			Error := FALSE;
		SF_MutingSeq_State#Muting_Backward_Start:
			MutingTimer(IN := FALSE);
			Ready := TRUE;
			S_AOPD_OUT := SAFEBOOL_Constant#SAFETRUE;
			S_MutingActive := SAFEBOOL_Constant#SAFEFALSE;
			SafetyDemand := FALSE;
			ResetRequest := FALSE;
			Error := FALSE;
		SF_MutingSeq_State#Muting_Backward_Active:
			MutingTimer(IN := TRUE, PT := MaxMutingTime);
			Ready := TRUE;
			S_AOPD_OUT := SAFEBOOL_Constant#SAFETRUE;
			S_MutingActive := SAFEBOOL_Constant#SAFETRUE;
			SafetyDemand := FALSE;
			ResetRequest := FALSE;
			Error := FALSE;
	ELSE
		ENO := FALSE;
	END_CASE;

	ENO := ENO AND CheckSAFEBOOL(S_AOPD_In) AND CheckSAFEBOOL(S_StartReset);

END_FUNCTION_BLOCK

/* returns a UINT value that can be added to the DiagCode indicating which muting states were active prior to the Error */
FUNCTION MutingSeqGetErrorStateOfMutingSensors : UINT
	VAR_INPUT
		MS_11 : BOOL;
		MS_12 : BOOL;
		MS_21 : BOOL;
		MS_22 : BOOL;
	END_VAR
	VAR
		Result : UINT := 16#0000;
	END_VAR
	IF(MS_11) THEN
		Result := Result + 16#0010;
	END_IF;
	IF(MS_12) THEN
		Result := Result + 16#0020;
	END_IF;
	IF(MS_21) THEN
		Result := Result + 16#0040;
	END_IF;
	IF(MS_22) THEN
		Result := Result + 16#0080;
	END_IF;

	MutingSeqGetErrorStateOfMutingSensors := Result;
END_FUNCTION

END_NAMESPACE
END_NAMESPACE

(* ---- SF_OutControl.iecst ---- *)
USING logicals.web.standard.safe;

NAMESPACE logicals.web.standard.safe
NAMESPACE plcopen

TYPE
	SF_OutControl_State : UINT(
	/* Static Reset signal in state 8401. */
	Reset_Error_1 := 16#C001,
	/* Static Reset signal in state 8404. */
	Reset_Error_2 := 16#C011,
	/* Static signal at ProcessControl in state 8006. */
	Control_Error := 16#C010,
	/* Simultaneous rising trigger at Reset and ProcessControl in state 8401. */
	Init_Error := 16#C020,
	/* Simultaneous rising trigger at Reset and ProcessControl in state 8404. */
	Lock_Error := 16#C030,
	/* The function block is not active (initial state). */
	Idle := 16#0000,
	/* Block activation startup inhibit is active. Reset required. */
	Init := 16#8401,
	/* Triggered safety function. */
	Safe := 16#8802,
	/* Safety function startup inhibit is active. Reset required. */
	Lock := 16#8404,
	/* Process control is not active. */
	Output_Disable := 16#8006,
	/* Process control is active and safety is enabled. */
	Output_Enable := 16#8000
	);
END_TYPE

/* Control of a safety output with a signal from the functional application and a safety signal with optional startup inhibits. */
FUNCTION_BLOCK SF_OutControl
	{ altName:="SF_OutControl"; bgColor:="Gold"; width:=360; }
	VAR_INPUT
		/* See Section 5.1.1 General Input Parameters */
		Activate : BOOL := FALSE;
		/* Variable.
		 * Control signal of the preceding safety FB.
		 * Typical function block signals from the library (e.g., SF_EStop, SF_GuardMonitoring, SF_TwoHand_Control_TypeII, and/or others).
		 * FALSE: The preceding safety FB's are in safe state.
		 * TRUE: The preceding safety FB's enable safety control. */
		S_SafeControl : SAFEBOOL := SAFEBOOL_Constant#SAFEFALSE;
		/* Variable or constant.
		 * Control signal from the functional application.
		 * FALSE: Request to set S_OutControl to FALSE.
		 * TRUE: Request to set S_OutControl to TRUE. */
		ProcessControl : BOOL := FALSE;
		/* Constant.
		 * Optional conditions for process control.
		 * FALSE: Dynamic change at ProcessControl (FALSE => TRUE) required after block activation or triggered safety function. Additional function start required.
		 * TRUE: No dynamic change at ProcessControl (FALSE => TRUE) required after block activation or triggered safety function. */
		StaticControl : BOOL := FALSE;
		/* See Section 5.1.1 General Input Parameters */
		S_StartReset : SAFEBOOL := SAFEBOOL_Constant#SAFEFALSE;
		/* See Section 5.1.1 General Input Parameters */
		S_AutoReset : SAFEBOOL := SAFEBOOL_Constant#SAFEFALSE;
		/* See Section 5.1.1 General Input Parameters */
		Reset : BOOL := FALSE;
	END_VAR

	VAR_OUTPUT
		/* See Section 5.1.2 General Output Parameters */
		Ready : BOOL := FALSE;
		/* Controls connected actuators.
		 * FALSE: Disable connected actuators.
		 * TRUE: Enable connected actuators. */
		S_OutControl : SAFEBOOL := SAFEBOOL_Constant#SAFEFALSE;
		/* See Section 5.1.2 General Output Parameters */
		SafetyDemand : BOOL := FALSE;
		/* See Section 5.1.2 General Output Parameters */
		ResetRequest : BOOL := FALSE;
		/* See Section 5.1.2 General Output Parameters */
		Error : BOOL := FALSE;
		/* See Section 5.1.2 General Output Parameters */
		DiagCode : WORD := 16#0000;
	END_VAR

	VAR
		R_Trig_Reset : R_TRIG;
		R_Trig_ProcessControl : R_TRIG;
	END_VAR

	R_Trig_Reset(Reset);
	R_Trig_ProcessControl(ProcessControl);

	IF(NOT Activate) THEN
		DiagCode := TO_WORD(SF_OutControl_State#Idle);
	ELSE
		CASE TO_UINT(DiagCode) OF
			SF_OutControl_State#Idle:
				/* IF(Activate) THEN - Active is always true here */
					DiagCode := TO_WORD(SF_OutControl_State#Init);
			SF_OutControl_State#Init:
				IF(Reset AND NOT R_Trig_Reset.Q AND NOT IS(S_StartReset)) THEN
					DiagCode := TO_WORD(SF_OutControl_State#Reset_Error_1);
				ELSIF(R_Trig_Reset.Q AND R_Trig_ProcessControl.Q) THEN
					DiagCode := TO_WORD(SF_OutControl_State#Init_Error);
				ELSIF(R_Trig_Reset.Q OR IS(S_StartReset)) THEN
					DiagCode := TO_WORD(SF_OutControl_State#Output_Disable);
				END_IF;
			SF_OutControl_State#Reset_Error_1:
				IF(NOT Reset) THEN
					DiagCode := TO_WORD(SF_OutControl_State#Init);
				END_IF;
			SF_OutControl_State#Init_Error:
				IF(NOT Reset) THEN
					DiagCode := TO_WORD(SF_OutControl_State#Init);
				END_IF;
			SF_OutControl_State#Output_Disable:
				IF(IS_NOT(S_SafeControl)) THEN
					DiagCode := TO_WORD(SF_OutControl_State#Safe);
				ELSIF(NOT R_Trig_ProcessControl.Q AND ProcessControl AND NOT StaticControl) THEN
					DiagCode := TO_WORD(SF_OutControl_State#Control_Error);
				ELSIF(IS(S_SafeControl) AND (R_Trig_ProcessControl.Q OR (StaticControl AND ProcessControl))) THEN
					DiagCode := TO_WORD(SF_OutControl_State#Output_Enable);
				END_IF;
			SF_OutControl_State#Control_Error:
				IF(NOT ProcessControl) THEN
					DiagCode := TO_WORD(SF_OutControl_State#Output_Disable);
				END_IF;
			SF_OutControl_State#Output_Enable:
				IF(IS_NOT(S_SafeControl)) THEN
					DiagCode := TO_WORD(SF_OutControl_State#Safe);
				ELSIF(NOT ProcessControl) THEN
					DiagCode := TO_WORD(SF_OutControl_State#Output_Disable);
				END_IF;
			SF_OutControl_State#Safe:
				IF(IS(S_SafeControl)) THEN
					DiagCode := TO_WORD(SF_OutControl_State#Lock);
				END_IF;
			SF_OutControl_State#Lock:
				IF(IS_NOT(S_SafeControl)) THEN
					DiagCode := TO_WORD(SF_OutControl_State#Safe);
				ELSIF(Reset AND NOT R_Trig_Reset.Q AND IS_NOT(S_AutoReset)) THEN
					DiagCode := TO_WORD(SF_OutControl_State#Reset_Error_2);
				ELSIF(R_Trig_Reset.Q AND R_Trig_ProcessControl.Q) THEN
					DiagCode := TO_WORD(SF_OutControl_State#Lock_Error);
				ELSIF(R_Trig_Reset.Q OR IS(S_AutoReset)) THEN
					DiagCode := TO_WORD(SF_OutControl_State#Output_Disable);
				END_IF;
			SF_OutControl_State#Lock_Error:
				IF(NOT Reset) THEN
					DiagCode := TO_WORD(SF_OutControl_State#Lock);
				END_IF;
			SF_OutControl_State#Reset_Error_2:
				IF(NOT Reset) THEN
					DiagCode := TO_WORD(SF_OutControl_State#Lock);
				END_IF;
		END_CASE;
	END_IF;

	CASE TO_UINT(DiagCode) OF
		SF_OutControl_State#Idle:
			Ready := FALSE;
			S_OutControl := SAFEBOOL_Constant#SAFEFALSE;
			SafetyDemand := FALSE;
			ResetRequest := FALSE;
			Error := FALSE;
		SF_OutControl_State#Init,
		SF_OutControl_State#Lock:
			Ready := TRUE;
			S_OutControl := SAFEBOOL_Constant#SAFEFALSE;
			SafetyDemand := FALSE;
			ResetRequest := TRUE;
			Error := FALSE;
		SF_OutControl_State#Safe:
			Ready := TRUE;
			S_OutControl := SAFEBOOL_Constant#SAFEFALSE;
			SafetyDemand := TRUE;
			ResetRequest := FALSE;
			Error := FALSE;
		SF_OutControl_State#Output_Disable:
			Ready := TRUE;
			S_OutControl := SAFEBOOL_Constant#SAFEFALSE;
			SafetyDemand := FALSE;
			ResetRequest := FALSE;
			Error := FALSE;
		SF_OutControl_State#Output_Enable:
			Ready := TRUE;
			S_OutControl := SAFEBOOL_Constant#SAFETRUE;
			SafetyDemand := FALSE;
			ResetRequest := FALSE;
			Error := FALSE;
		SF_OutControl_State#Reset_Error_1,
		SF_OutControl_State#Reset_Error_2,
		SF_OutControl_State#Control_Error,
		SF_OutControl_State#Init_Error,
		SF_OutControl_State#Lock_Error:
			Ready := TRUE;
			S_OutControl := SAFEBOOL_Constant#SAFEFALSE;
			SafetyDemand := FALSE;
			ResetRequest := FALSE;
			Error := TRUE;
	END_CASE;

	ENO := ENO AND CheckSAFEBOOL(S_SafeControl) AND CheckSAFEBOOL(S_StartReset) AND CheckSAFEBOOL(S_AutoReset);

END_FUNCTION_BLOCK

END_NAMESPACE
END_NAMESPACE

(* ---- SF_Override.iecst ---- *)
USING logicals.web.standard.safe;

NAMESPACE logicals.web.standard.safe
NAMESPACE plcopen

TYPE
	SF_Override_State : UINT(
		/* The function block is not active (initial state). */
		Idle := 16#0000,
		/* Static Reset condition detected after FB activation. */
		Reset_Error := 16#C011,
		/* Max Override time elapsed. */
		Override_Error := 16#C410,
		/* Protection field interrupted and muting not active or override is not active
		 * and the timer for the MaxOverrideTime will be reset. */
		Safety_Demand_AOPD := 16#8002,
		/* The pre-connected muting FB shows an error but the safeguard (e.g. light
		 * curtain) is not interrupted and no muting sensor is blocked. */
		Muting_Error_but_Override_not_possible := 16#8012,
		/* The pre-connected muting FB shows an error and the safeguard (e.g. light
		 * curtain) is interrupted and/or at least one muting sensor is blocked. */
		Override_Possible := 16#8022,
		/* The override start signal is set to FALSE during override process. The
		 * time for the MaxOverrideTime is still running. */
		Override_Interrupt := 16#8832,
		/* Override is active and the timer for the MaxOverrideTime is starting to run. */
		Override_Active := 16#8000,
		/* S_AOPD_Out from the pre-connected function block is TRUE. */
		AOPD_Free := 16#8100
	);
END_TYPE

FUNCTION_BLOCK SF_Override
	{ altName:="SF_Override"; bgColor:="Gold"; width:=360; }
	VAR_INPUT
		/* See Section 5.1.1 General Input Parameters */
		Activate : BOOL := FALSE;
		/* Variable. OSSD signal from AOPD.
		 * FALSE: Protection field interrupted.
		 * TRUE: Protection field not interrupted. */
		S_AOPD_In : SAFEBOOL := SAFEBOOL_Constant#SAFEFALSE;
		/* Variable. S_AOPD_OUT signal from the previous muting block.
		 * FALSE/TRUE: The Status of the Safety related output.
		 * S_AOPD_OUT from the previous muting block. */
		S_Muting_AOPD_Out : SAFEBOOL := SAFEBOOL_Constant#SAFEFALSE;
		/* Error output of the previous connected Muting-FB.
		 * FALSE: No error.
		 * TRUE: Error in Muting Process */
		MutingError : BOOL := FALSE;
		/* Variable.
		 * Status of the Muting sensor signal which is connected at the
		 * input MutingSwitch11 of the previous muting function block
		 * FALSE: Muting sensor 11 not actuated.
		 * TRUE: Workpiece actuates muting sensor 11. */
		MutingSwitch11 : BOOL := FALSE;
		/* Variable.
		 * Status of the Muting sensor signal which is connected at the
		 * input MutingSwitch12 of the previous muting function block
		 * FALSE: Muting sensor 12 not actuated.
		 * TRUE: Workpiece actuates muting sensor 12. */
		MutingSwitch12 : BOOL := FALSE;
		/* Variable.
		 * Status of the Muting sensor signal which is connected at the
		 * input MutingSwitch21 of the previous muting function block
		 * FALSE: Muting sensor 21 not actuated.
		 * TRUE: Workpiece actuates muting sensor 21.
		 * It shall be noted that this parameter is not connected if the
		 * previous muting function is the SF_MutingPar_2Sensor. */
		MutingSwitch21 : BOOL := FALSE;
		/* Variable.
		 * Status of the Muting sensor signal which is connected at the
		 * input MutingSwitch22 of the previous muting function block
		 * FALSE: Muting sensor 22 not actuated.
		 * TRUE: Workpiece actuates muting sensor 22.
		 * It shall be noted that this parameter is not connected if the
		 * previous muting function is the SF_MutingPar_2Sensor. */
		MutingSwitch22 : BOOL := FALSE;
		/* Constant 0..10 min;
		 * Maximum time for the overall Override process.
		 * The time is started when the start conditions for the override
		 * process are available. The timer is stopped when all the muting
		 * sensors are not muted anymore.
		 */
		MaxOverrideTime : TIME := T#0s;
		/* Signal for the start and stop of override functionality.
		 * A rising edge is needed to start hte override functionality.
		 * TRUE: If all override conditions are fulfilled, the override process
		 * starts. At this moment also the time for the MaxOverrideTime starts.
		 * FALSE: THe override process stops. The timer for the MaxOverrideTime
		 * continues till the muting process is finished (transition 8832 to 8802).
		 */
		S_StartStopOverride : SAFEBOOL := SAFEBOOL_Constant#SAFEFALSE;
		/* See 5.1.1 General Input Parameters */
		Reset : BOOL := FALSE;
	END_VAR
	VAR_OUTPUT
		/* See 5.1.2 General Output Parameters */
		Ready : BOOL := FALSE;
		/* Safety related output, indicates status of the muted guard or
		 * override signal.
		 * FALSE: AOPD protection field interrupted and muting not
		 * active or override is not active.
		 * TRUE: AOPD protection field not interrupted or muting active
		 * or override is active. */
		S_AOPD_OUT : SAFEBOOL := SAFEBOOL_Constant#SAFEFALSE;
		/* Status signaling that override is possible
		 * FALSE: Override not possible
		 * TRUE: Override possible */
		OverridePossible : BOOL := FALSE;
		/* Indicates the status of Override process.
		 * FALSE: Override not active.
		 * TRUE: Override active. */
		OverrideActive : BOOL := FALSE;
		/* See 5.1.2 General Output Parameters */
		SafetyDemand : BOOL := FALSE;
		/* See 5.1.2 General Output Parameters */
		ResetRequest : BOOL := FALSE;
		/* See 5.1.2 General Output Parameters */
		Error : BOOL := FALSE;
		/* See 5.1.2 General Output Parameters */
		DiagCode : WORD := 16#0000;
	END_VAR
	VAR
		OverrideTimer : TON;
		AnySwitchActive : BOOL;
		R_Trig_StartStopOverride : R_TRIG;
		R_Trig_Reset : R_TRIG;
	END_VAR

	IF(NOT Activate) THEN
		DiagCode := TO_WORD(SF_Override_State#Idle);
	ELSE
		AnySwitchActive := MutingSwitch11 OR MutingSwitch12 OR MutingSwitch21 OR MutingSwitch22;
		R_Trig_StartStopOverride(IS(S_StartStopOverride));
		R_Trig_Reset(Reset);

		CASE TO_UINT(DiagCode) OF
			SF_Override_State#Idle:
				// Activate is always true here
				DiagCode := TO_WORD(SF_Override_State#Safety_Demand_AOPD);
			SF_Override_State#Safety_Demand_AOPD:
				IF(MutingError AND (IS(S_AOPD_In) AND NOT AnySwitchActive)) THEN
					DiagCode := TO_WORD(SF_Override_State#Muting_Error_but_Override_not_possible);
				ELSIF(MutingError AND (IS_NOT(S_AOPD_In) OR AnySwitchActive)) THEN
					DiagCode := TO_WORD(SF_Override_State#Override_Possible);
				ELSIF(IS(S_Muting_AOPD_Out)) THEN
					DiagCode := TO_WORD(SF_Override_State#AOPD_Free);
				END_IF;
			SF_Override_State#Override_Possible:
				IF(NOT (MutingError AND (IS_NOT(S_AOPD_In) OR AnySwitchActive))) THEN
					DiagCode := TO_WORD(SF_Override_State#Safety_Demand_AOPD);
				ELSIF(R_Trig_StartStopOverride.Q) THEN
					DiagCode := TO_WORD(SF_Override_State#Override_Active);
				END_IF;
			SF_Override_State#Override_Active:
				IF(OverrideTimer.Q) THEN
					DiagCode := TO_WORD(SF_Override_State#Override_Error);
				ELSIF(IS_NOT(S_StartStopOverride)) THEN
					DiagCode := TO_WORD(SF_Override_State#Override_Interrupt);
				ELSIF(NOT(MutingError AND (IS_NOT(S_AOPD_In) OR AnySwitchActive))) THEN
					DiagCode := TO_WORD(SF_Override_State#Safety_Demand_AOPD);
				END_IF;
			SF_Override_State#Override_Interrupt:
				IF(OverrideTimer.Q) THEN
					DiagCode := TO_WORD(SF_Override_State#Override_Error);
				ELSIF(NOT(MutingError AND (IS_NOT(S_AOPD_In) OR AnySwitchActive))) THEN
					DiagCode := TO_WORD(SF_Override_State#Safety_Demand_AOPD);
				ELSIF(IS(S_StartStopOverride)) THEN
					DiagCode := TO_WORD(SF_Override_State#Override_Active);
				END_IF;
			SF_Override_State#Override_Error:
				IF(Reset AND NOT R_Trig_Reset.Q) THEN
					DiagCode := TO_WORD(SF_Override_State#Reset_Error);
				ELSIF(R_Trig_Reset.Q) THEN
					DiagCode := TO_WORD(SF_Override_State#Safety_Demand_AOPD);
				END_IF;
			SF_Override_State#Reset_Error:
				IF(NOT Reset) THEN
					DiagCode := TO_WORD(SF_Override_State#Override_Error);
				END_IF;
			SF_Override_State#AOPD_Free:
				IF(IS_NOT(S_Muting_AOPD_Out)) THEN
					DiagCode := TO_WORD(SF_Override_State#Safety_Demand_AOPD);
				END_IF;
			SF_Override_State#Muting_Error_but_Override_not_possible:
				IF(NOT MutingError) THEN
					DiagCode := TO_WORD(SF_Override_State#Safety_Demand_AOPD);
				END_IF;
		ELSE
				ENO := FALSE;
		END_CASE;
	END_IF;

	CASE TO_UINT(DiagCode) OF
		SF_Override_State#Idle:
			OverrideTimer(IN := FALSE);
			Ready := FALSE;
			S_AOPD_OUT := SAFEBOOL_Constant#SAFEFALSE;
			OverridePossible := FALSE;
			OverrideActive := FALSE;
			SafetyDemand := FALSE;
			ResetRequest := FALSE;
			Error := FALSE;
		SF_Override_State#Reset_Error:
			OverrideTimer(IN := FALSE);
			Ready := TRUE;
			S_AOPD_OUT := SAFEBOOL_Constant#SAFEFALSE;
			OverridePossible := FALSE;
			OverrideActive := FALSE;
			SafetyDemand := FALSE;
			ResetRequest := FALSE;
			Error := TRUE;
		SF_Override_State#Override_Error:
			OverrideTimer(IN := FALSE);
			Ready := TRUE;
			S_AOPD_OUT := SAFEBOOL_Constant#SAFEFALSE;
			OverridePossible := FALSE;
			OverrideActive := FALSE;
			SafetyDemand := FALSE;
			ResetRequest := TRUE;
			Error := TRUE;
		SF_Override_State#Safety_Demand_AOPD:
			OverrideTimer(IN := FALSE);
			Ready := TRUE;
			S_AOPD_OUT := SAFEBOOL_Constant#SAFEFALSE;
			OverridePossible := FALSE;
			OverrideActive := FALSE;
			SafetyDemand := FALSE;
			ResetRequest := FALSE;
			Error := FALSE;
		SF_Override_State#Muting_Error_but_Override_not_possible:
			OverrideTimer(IN := FALSE);
			Ready := TRUE;
			S_AOPD_OUT := SAFEBOOL_Constant#SAFEFALSE;
			OverridePossible := FALSE;
			OverrideActive := FALSE;
			SafetyDemand := FALSE;
			ResetRequest := FALSE;
			Error := FALSE;
		SF_Override_State#Override_Possible:
			OverrideTimer(IN := FALSE);
			Ready := TRUE;
			S_AOPD_OUT := SAFEBOOL_Constant#SAFEFALSE;
			OverridePossible := TRUE;
			OverrideActive := FALSE;
			SafetyDemand := FALSE;
			ResetRequest := FALSE;
			Error := FALSE;
		SF_Override_State#Override_Interrupt:
			OverrideTimer(IN := TRUE, PT := MaxOverrideTime);
			Ready := TRUE;
			S_AOPD_OUT := SAFEBOOL_Constant#SAFEFALSE;
			OverridePossible := TRUE;
			OverrideActive := FALSE;
			SafetyDemand := TRUE;
			ResetRequest := FALSE;
			Error := FALSE;
		SF_Override_State#Override_Active:
			OverrideTimer(IN := TRUE, PT := MaxOverrideTime);
			Ready := TRUE;
			S_AOPD_OUT := SAFEBOOL_Constant#SAFETRUE;
			OverridePossible := TRUE;
			OverrideActive := TRUE;
			SafetyDemand := FALSE;
			ResetRequest := FALSE;
			Error := FALSE;
		SF_Override_State#AOPD_Free:
			OverrideTimer(IN := FALSE);
			Ready := TRUE;
			S_AOPD_OUT := SAFEBOOL_Constant#SAFETRUE;
			OverridePossible := FALSE;
			OverrideActive := FALSE;
			SafetyDemand := FALSE;
			ResetRequest := FALSE;
			Error := FALSE;
		ELSE
			ENO := FALSE;
	END_CASE;

	ENO := ENO AND CheckSAFEBOOL(S_AOPD_In) AND CheckSAFEBOOL(S_Muting_AOPD_Out) AND CheckSAFEBOOL(S_StartStopOverride);

END_FUNCTION_BLOCK

END_NAMESPACE
END_NAMESPACE
